  PROC DrawPart46()
    MoveL Offs(pOrigin,252.98,111.04,0.00),v40,z0,tPen\WObj:=wPaper;
    MoveL Offs(pOrigin,252.55,110.82,0.00),v40,fine,tPen\WObj:=wPaper;
    MoveL Offs(pOrigin,252.55,110.82,6.00),v60,z5,tPen\WObj:=wPaper;
    MoveL Offs(pOrigin,253.40,114.65,6.00),vTravel,z5,tPen\WObj:=wPaper;
    MoveL Offs(pOrigin,253.40,114.65,0.00),v60,z0,tPen\WObj:=wPaper;
    MoveL Offs(pOrigin,252.98,115.29,0.00),v40,z0,tPen\WObj:=wPaper;
    MoveL Offs(pOrigin,253.40,114.65,0.00),v40,fine,tPen\WObj:=wPaper;
    MoveL Offs(pOrigin,253.40,114.65,6.00),v60,z5,tPen\WObj:=wPaper;
    MoveL Offs(pOrigin,248.51,114.22,6.00),vTravel,z5,tPen\WObj:=wPaper;
    MoveL Offs(pOrigin,248.51,114.22,0.00),v60,z0,tPen\WObj:=wPaper;
    MoveL Offs(pOrigin,248.73,114.65,0.00),v40,z0,tPen\WObj:=wPaper;
    MoveL Offs(pOrigin,248.51,114.22,0.00),v40,fine,tPen\WObj:=wPaper;
    MoveL Offs(pOrigin,248.51,114.22,6.00),v60,z5,tPen\WObj:=wPaper;
    MoveL Offs(pOrigin,237.25,127.61,6.00),vTravel,z5,tPen\WObj:=wPaper;
    MoveL Offs(pOrigin,237.25,127.61,0.00),v60,z0,tPen\WObj:=wPaper;
    MoveL Offs(pOrigin,235.55,135.69,0.00),v40,fine,tPen\WObj:=wPaper;
    MoveL Offs(pOrigin,235.55,135.69,6.00),v60,z5,tPen\WObj:=wPaper;
    MoveL Offs(pOrigin,208.14,123.79,6.00),vTravel,z5,tPen\WObj:=wPaper;
    MoveL Offs(pOrigin,208.14,123.79,0.00),v60,z0,tPen\WObj:=wPaper;
    MoveL Offs(pOrigin,208.92,123.36,0.00),v40,z0,tPen\WObj:=wPaper;
    MoveL Offs(pOrigin,211.75,113.38,0.00),v40,z0,tPen\WObj:=wPaper;
    MoveL Offs(pOrigin,214.73,101.05,0.00),v40,z0,tPen\WObj:=wPaper;
    MoveL Offs(pOrigin,216.43,90.85,0.00),v40,z0,tPen\WObj:=wPaper;
    MoveL Offs(pOrigin,217.27,82.14,0.00),v40,z0,tPen\WObj:=wPaper;
    MoveL Offs(pOrigin,217.49,71.94,0.00),v40,z0,tPen\WObj:=wPaper;
    MoveL Offs(pOrigin,216.85,63.44,0.00),v40,z0,tPen\WObj:=wPaper;
    MoveL Offs(pOrigin,216.00,62.80,0.00),v40,z0,tPen\WObj:=wPaper;
    MoveL Offs(pOrigin,216.00,62.80,0.00),v40,z0,tPen\WObj:=wPaper;
    MoveL Offs(pOrigin,215.15,64.07,0.00),v40,z0,tPen\WObj:=wPaper;
    MoveL Offs(pOrigin,215.15,68.11,0.00),v40,z0,tPen\WObj:=wPaper;
    MoveL Offs(pOrigin,214.58,70.45,0.00),v40,z0,tPen\WObj:=wPaper;
    MoveL Offs(pOrigin,213.66,71.94,0.00),v40,z0,tPen\WObj:=wPaper;
    MoveL Offs(pOrigin,212.39,72.86,0.00),v40,z0,tPen\WObj:=wPaper;
    MoveL Offs(pOrigin,207.71,74.70,0.00),v40,z0,tPen\WObj:=wPaper;
    MoveL Offs(pOrigin,204.31,75.34,0.00),v40,z0,tPen\WObj:=wPaper;
    MoveL Offs(pOrigin,198.36,75.76,0.00),v40,z0,tPen\WObj:=wPaper;
    MoveL Offs(pOrigin,195.60,75.55,0.00),v40,z0,tPen\WObj:=wPaper;
    MoveL Offs(pOrigin,195.60,75.55,0.00),v40,z0,tPen\WObj:=wPaper;
    MoveL Offs(pOrigin,196.59,73.21,0.00),v40,z0,tPen\WObj:=wPaper;
    MoveL Offs(pOrigin,196.24,72.79,0.00),v40,z0,tPen\WObj:=wPaper;
    MoveL Offs(pOrigin,194.96,72.93,0.00),v40,z0,tPen\WObj:=wPaper;
    MoveL Offs(pOrigin,192.20,74.70,0.00),v40,z0,tPen\WObj:=wPaper;
    MoveL Offs(pOrigin,192.20,74.70,0.00),v40,z0,tPen\WObj:=wPaper;
    MoveL Offs(pOrigin,192.06,75.76,0.00),v40,z0,tPen\WObj:=wPaper;
    MoveL Offs(pOrigin,189.23,78.31,0.00),v40,z0,tPen\WObj:=wPaper;
    MoveL Offs(pOrigin,189.23,78.31,0.00),v40,z0,tPen\WObj:=wPaper;
    MoveL Offs(pOrigin,187.52,76.47,0.00),v40,z0,tPen\WObj:=wPaper;
    MoveL Offs(pOrigin,186.25,76.82,0.00),v40,fine,tPen\WObj:=wPaper;
    MoveL Offs(pOrigin,186.25,76.82,6.00),v60,z5,tPen\WObj:=wPaper;
    MoveL Offs(pOrigin,187.74,76.40,6.00),vTravel,z5,tPen\WObj:=wPaper;
    MoveL Offs(pOrigin,187.74,76.40,0.00),v60,z0,tPen\WObj:=wPaper;
    MoveL Offs(pOrigin,187.95,76.05,0.00),v40,z0,tPen\WObj:=wPaper;
    MoveL Offs(pOrigin,190.71,74.84,0.00),v40,z0,tPen\WObj:=wPaper;
    MoveL Offs(pOrigin,192.20,74.70,0.00),v40,fine,tPen\WObj:=wPaper;
    MoveL Offs(pOrigin,192.20,74.70,6.00),v60,z5,tPen\WObj:=wPaper;
    MoveL Offs(pOrigin,190.50,75.12,6.00),vTravel,z5,tPen\WObj:=wPaper;
    MoveL Offs(pOrigin,190.50,75.12,0.00),v60,z0,tPen\WObj:=wPaper;
    MoveL Offs(pOrigin,190.93,74.91,0.00),v40,z0,tPen\WObj:=wPaper;
    MoveL Offs(pOrigin,190.50,75.12,0.00),v40,z0,tPen\WObj:=wPaper;
    MoveL Offs(pOrigin,189.44,75.55,0.00),v40,z0,tPen\WObj:=wPaper;
    MoveL Offs(pOrigin,189.86,75.34,0.00),v40,z0,tPen\WObj:=wPaper;
    MoveL Offs(pOrigin,189.44,75.55,0.00),v40,fine,tPen\WObj:=wPaper;
    MoveL Offs(pOrigin,189.44,75.55,6.00),v60,z5,tPen\WObj:=wPaper;
    MoveL Offs(pOrigin,190.29,77.46,6.00),vTravel,z5,tPen\WObj:=wPaper;
    MoveL Offs(pOrigin,190.29,77.46,0.00),v60,z0,tPen\WObj:=wPaper;
    MoveL Offs(pOrigin,190.50,77.04,0.00),v40,z0,tPen\WObj:=wPaper;
    MoveL Offs(pOrigin,190.29,77.46,0.00),v40,z0,tPen\WObj:=wPaper;
    MoveL Offs(pOrigin,189.86,77.68,0.00),v40,z0,tPen\WObj:=wPaper;
    MoveL Offs(pOrigin,189.65,78.10,0.00),v40,z0,tPen\WObj:=wPaper;
    MoveL Offs(pOrigin,189.86,77.68,0.00),v40,fine,tPen\WObj:=wPaper;
    MoveL Offs(pOrigin,189.86,77.68,6.00),v60,z5,tPen\WObj:=wPaper;
    MoveL Offs(pOrigin,189.23,78.74,6.00),vTravel,z5,tPen\WObj:=wPaper;
    MoveL Offs(pOrigin,189.23,78.74,0.00),v60,z0,tPen\WObj:=wPaper;
    MoveL Offs(pOrigin,187.52,80.44,0.00),v40,z0,tPen\WObj:=wPaper;
    MoveL Offs(pOrigin,187.52,80.44,0.00),v40,z0,tPen\WObj:=wPaper;
    MoveL Offs(pOrigin,188.38,81.71,0.00),v40,z0,tPen\WObj:=wPaper;
    MoveL Offs(pOrigin,188.16,82.35,0.00),v40,z0,tPen\WObj:=wPaper;
    MoveL Offs(pOrigin,187.95,82.78,0.00),v40,z0,tPen\WObj:=wPaper;
    MoveL Offs(pOrigin,188.16,82.35,0.00),v40,z0,tPen\WObj:=wPaper;
    MoveL Offs(pOrigin,187.52,82.99,0.00),v40,z0,tPen\WObj:=wPaper;
    MoveL Offs(pOrigin,187.31,83.41,0.00),v40,z0,tPen\WObj:=wPaper;
    MoveL Offs(pOrigin,187.52,82.99,0.00),v40,fine,tPen\WObj:=wPaper;
    MoveL Offs(pOrigin,187.52,82.99,6.00),v60,z5,tPen\WObj:=wPaper;
    MoveL Offs(pOrigin,186.46,84.05,6.00),vTravel,z5,tPen\WObj:=wPaper;
    MoveL Offs(pOrigin,186.46,84.05,0.00),v60,z0,tPen\WObj:=wPaper;
    MoveL Offs(pOrigin,186.89,83.62,0.00),v40,z0,tPen\WObj:=wPaper;
    MoveL Offs(pOrigin,186.46,84.05,0.00),v40,z0,tPen\WObj:=wPaper;
    MoveL Offs(pOrigin,186.04,84.26,0.00),v40,z0,tPen\WObj:=wPaper;
    MoveL Offs(pOrigin,185.82,84.69,0.00),v40,z0,tPen\WObj:=wPaper;
    MoveL Offs(pOrigin,186.04,84.26,0.00),v40,fine,tPen\WObj:=wPaper;
    MoveL Offs(pOrigin,186.04,84.26,6.00),v60,z5,tPen\WObj:=wPaper;
    MoveL Offs(pOrigin,184.55,83.20,6.00),vTravel,z5,tPen\WObj:=wPaper;
    MoveL Offs(pOrigin,184.55,83.20,0.00),v60,z0,tPen\WObj:=wPaper;
    MoveL Offs(pOrigin,187.52,80.44,0.00),v40,fine,tPen\WObj:=wPaper;
    MoveL Offs(pOrigin,187.52,80.44,6.00),v60,z5,tPen\WObj:=wPaper;
    MoveL Offs(pOrigin,188.16,79.38,6.00),vTravel,z5,tPen\WObj:=wPaper;
    MoveL Offs(pOrigin,188.16,79.38,0.00),v60,z0,tPen\WObj:=wPaper;
    MoveL Offs(pOrigin,187.74,80.01,0.00),v40,z0,tPen\WObj:=wPaper;
    MoveL Offs(pOrigin,188.16,79.38,0.00),v40,fine,tPen\WObj:=wPaper;
    MoveL Offs(pOrigin,188.16,79.38,6.00),v60,z5,tPen\WObj:=wPaper;
    MoveL Offs(pOrigin,189.23,78.74,6.00),vTravel,z5,tPen\WObj:=wPaper;
    MoveL Offs(pOrigin,189.23,78.74,0.00),v60,z0,tPen\WObj:=wPaper;
    MoveL Offs(pOrigin,189.86,79.38,0.00),v40,z0,tPen\WObj:=wPaper;
    MoveL Offs(pOrigin,189.65,80.44,0.00),v40,z0,tPen\WObj:=wPaper;
    MoveL Offs(pOrigin,189.44,80.86,0.00),v40,z0,tPen\WObj:=wPaper;
    MoveL Offs(pOrigin,189.65,80.44,0.00),v40,fine,tPen\WObj:=wPaper;
    MoveL Offs(pOrigin,189.65,80.44,6.00),v60,z5,tPen\WObj:=wPaper;
    MoveL Offs(pOrigin,192.20,77.68,6.00),vTravel,z5,tPen\WObj:=wPaper;
    MoveL Offs(pOrigin,192.20,77.68,0.00),v60,z0,tPen\WObj:=wPaper;
    MoveL Offs(pOrigin,191.56,78.31,0.00),v40,z0,tPen\WObj:=wPaper;
    MoveL Offs(pOrigin,192.20,77.68,0.00),v40,fine,tPen\WObj:=wPaper;
    MoveL Offs(pOrigin,192.20,77.68,6.00),v60,z5,tPen\WObj:=wPaper;
    MoveL Offs(pOrigin,193.90,76.19,6.00),vTravel,z5,tPen\WObj:=wPaper;
    MoveL Offs(pOrigin,193.90,76.19,0.00),v60,z0,tPen\WObj:=wPaper;
    MoveL Offs(pOrigin,193.05,77.04,0.00),v40,z0,tPen\WObj:=wPaper;
    MoveL Offs(pOrigin,193.90,76.19,0.00),v40,fine,tPen\WObj:=wPaper;
    MoveL Offs(pOrigin,193.90,76.19,6.00),v60,z5,tPen\WObj:=wPaper;
    MoveL Offs(pOrigin,185.19,82.56,6.00),vTravel,z5,tPen\WObj:=wPaper;
    MoveL Offs(pOrigin,185.19,82.56,0.00),v60,z0,tPen\WObj:=wPaper;
    MoveL Offs(pOrigin,185.40,82.14,0.00),v40,z0,tPen\WObj:=wPaper;
  ENDPROC

  PROC DrawPart47()
    MoveL Offs(pOrigin,185.19,82.56,0.00),v40,fine,tPen\WObj:=wPaper;
    MoveL Offs(pOrigin,185.19,82.56,6.00),v60,z5,tPen\WObj:=wPaper;
    MoveL Offs(pOrigin,184.12,83.41,6.00),vTravel,z5,tPen\WObj:=wPaper;
    MoveL Offs(pOrigin,184.12,83.41,0.00),v60,z0,tPen\WObj:=wPaper;
    MoveL Offs(pOrigin,179.24,87.88,0.00),v40,z0,tPen\WObj:=wPaper;
    MoveL Offs(pOrigin,169.46,95.95,0.00),v40,z0,tPen\WObj:=wPaper;
    MoveL Offs(pOrigin,169.46,95.95,0.00),v40,z0,tPen\WObj:=wPaper;
    MoveL Offs(pOrigin,168.82,95.31,0.00),v40,fine,tPen\WObj:=wPaper;
    MoveL Offs(pOrigin,168.82,95.31,6.00),v60,z5,tPen\WObj:=wPaper;
    MoveL Offs(pOrigin,169.68,96.59,6.00),vTravel,z5,tPen\WObj:=wPaper;
    MoveL Offs(pOrigin,169.68,96.59,0.00),v60,z0,tPen\WObj:=wPaper;
    MoveL Offs(pOrigin,167.98,97.22,0.00),v40,z0,tPen\WObj:=wPaper;
    MoveL Offs(pOrigin,166.91,96.80,0.00),v40,z0,tPen\WObj:=wPaper;
    MoveL Offs(pOrigin,165.64,95.53,0.00),v40,fine,tPen\WObj:=wPaper;
    MoveL Offs(pOrigin,165.64,95.53,6.00),v60,z5,tPen\WObj:=wPaper;
    MoveL Offs(pOrigin,163.51,97.01,6.00),vTravel,z5,tPen\WObj:=wPaper;
    MoveL Offs(pOrigin,163.51,97.01,0.00),v60,z0,tPen\WObj:=wPaper;
    MoveL Offs(pOrigin,162.80,95.74,0.00),v40,z0,tPen\WObj:=wPaper;
    MoveL Offs(pOrigin,162.38,93.82,0.00),v40,z0,tPen\WObj:=wPaper;
    MoveL Offs(pOrigin,161.46,93.19,0.00),v40,z0,tPen\WObj:=wPaper;
    MoveL Offs(pOrigin,160.96,92.34,0.00),v40,z0,tPen\WObj:=wPaper;
    MoveL Offs(pOrigin,160.96,92.34,0.00),v40,z0,tPen\WObj:=wPaper;
    MoveL Offs(pOrigin,158.20,91.28,0.00),v40,z0,tPen\WObj:=wPaper;
    MoveL Offs(pOrigin,155.01,92.48,0.00),v40,z0,tPen\WObj:=wPaper;
    MoveL Offs(pOrigin,151.40,94.68,0.00),v40,fine,tPen\WObj:=wPaper;
    MoveL Offs(pOrigin,151.40,94.68,6.00),v60,z5,tPen\WObj:=wPaper;
    MoveL Offs(pOrigin,146.51,99.56,6.00),vTravel,z5,tPen\WObj:=wPaper;
    MoveL Offs(pOrigin,146.51,99.56,0.00),v60,z0,tPen\WObj:=wPaper;
    MoveL Offs(pOrigin,151.61,98.93,0.00),v40,z0,tPen\WObj:=wPaper;
    MoveL Offs(pOrigin,157.99,98.93,0.00),v40,z0,tPen\WObj:=wPaper;
    MoveL Offs(pOrigin,160.54,99.49,0.00),v40,z0,tPen\WObj:=wPaper;
    MoveL Offs(pOrigin,162.88,101.90,0.00),v40,z0,tPen\WObj:=wPaper;
    MoveL Offs(pOrigin,162.88,101.90,0.00),v40,z0,tPen\WObj:=wPaper;
    MoveL Offs(pOrigin,161.81,101.05,0.00),v40,fine,tPen\WObj:=wPaper;
    MoveL Offs(pOrigin,161.81,101.05,6.00),v60,z5,tPen\WObj:=wPaper;
    MoveL Offs(pOrigin,162.88,103.18,6.00),vTravel,z5,tPen\WObj:=wPaper;
    MoveL Offs(pOrigin,162.88,103.18,0.00),v60,z0,tPen\WObj:=wPaper;
    MoveL Offs(pOrigin,160.96,103.74,0.00),v40,z0,tPen\WObj:=wPaper;
    MoveL Offs(pOrigin,159.26,104.95,0.00),v40,z0,tPen\WObj:=wPaper;
    MoveL Offs(pOrigin,156.50,106.22,0.00),v40,z0,tPen\WObj:=wPaper;
    MoveL Offs(pOrigin,150.76,107.85,0.00),v40,fine,tPen\WObj:=wPaper;
    MoveL Offs(pOrigin,150.76,107.85,6.00),v60,z5,tPen\WObj:=wPaper;
    MoveL Offs(pOrigin,143.96,115.07,6.00),vTravel,z5,tPen\WObj:=wPaper;
    MoveL Offs(pOrigin,143.96,115.07,0.00),v60,z0,tPen\WObj:=wPaper;
    MoveL Offs(pOrigin,148.85,116.35,0.00),v40,z0,tPen\WObj:=wPaper;
    MoveL Offs(pOrigin,152.04,116.78,0.00),v40,z0,tPen\WObj:=wPaper;
    MoveL Offs(pOrigin,155.65,116.56,0.00),v40,z0,tPen\WObj:=wPaper;
    MoveL Offs(pOrigin,158.20,115.78,0.00),v40,z0,tPen\WObj:=wPaper;
    MoveL Offs(pOrigin,158.84,115.29,0.00),v40,z0,tPen\WObj:=wPaper;
    MoveL Offs(pOrigin,159.48,115.07,0.00),v40,z0,tPen\WObj:=wPaper;
    MoveL Offs(pOrigin,159.26,115.29,0.00),v40,z0,tPen\WObj:=wPaper;
    MoveL Offs(pOrigin,159.48,114.86,0.00),v40,z0,tPen\WObj:=wPaper;
    MoveL Offs(pOrigin,161.18,114.44,0.00),v40,fine,tPen\WObj:=wPaper;
    MoveL Offs(pOrigin,161.18,114.44,6.00),v60,z5,tPen\WObj:=wPaper;
    MoveL Offs(pOrigin,165.21,112.74,6.00),vTravel,z5,tPen\WObj:=wPaper;
    MoveL Offs(pOrigin,165.21,112.74,0.00),v60,z0,tPen\WObj:=wPaper;
    MoveL Offs(pOrigin,165.43,113.16,0.00),v40,z0,tPen\WObj:=wPaper;
    MoveL Offs(pOrigin,165.21,112.74,0.00),v40,z0,tPen\WObj:=wPaper;
    MoveL Offs(pOrigin,165.64,113.59,0.00),v40,z0,tPen\WObj:=wPaper;
    MoveL Offs(pOrigin,165.85,114.01,0.00),v40,z0,tPen\WObj:=wPaper;
    MoveL Offs(pOrigin,165.64,113.59,0.00),v40,fine,tPen\WObj:=wPaper;
    MoveL Offs(pOrigin,165.64,113.59,6.00),v60,z5,tPen\WObj:=wPaper;
    MoveL Offs(pOrigin,166.27,114.65,6.00),vTravel,z5,tPen\WObj:=wPaper;
    MoveL Offs(pOrigin,166.27,114.65,0.00),v60,z0,tPen\WObj:=wPaper;
    MoveL Offs(pOrigin,166.49,115.07,0.00),v40,z0,tPen\WObj:=wPaper;
    MoveL Offs(pOrigin,166.27,114.65,0.00),v40,fine,tPen\WObj:=wPaper;
    MoveL Offs(pOrigin,166.27,114.65,6.00),v60,z5,tPen\WObj:=wPaper;
    MoveL Offs(pOrigin,169.25,113.38,6.00),vTravel,z5,tPen\WObj:=wPaper;
    MoveL Offs(pOrigin,169.25,113.38,0.00),v60,z0,tPen\WObj:=wPaper;
    MoveL Offs(pOrigin,169.68,114.01,0.00),v40,z0,tPen\WObj:=wPaper;
    MoveL Offs(pOrigin,169.25,113.38,0.00),v40,fine,tPen\WObj:=wPaper;
    MoveL Offs(pOrigin,169.25,113.38,6.00),v60,z5,tPen\WObj:=wPaper;
    MoveL Offs(pOrigin,168.19,111.89,6.00),vTravel,z5,tPen\WObj:=wPaper;
    MoveL Offs(pOrigin,168.19,111.89,0.00),v60,z0,tPen\WObj:=wPaper;
    MoveL Offs(pOrigin,168.61,112.53,0.00),v40,z0,tPen\WObj:=wPaper;
    MoveL Offs(pOrigin,168.19,111.89,0.00),v40,fine,tPen\WObj:=wPaper;
    MoveL Offs(pOrigin,168.19,111.89,6.00),v60,z5,tPen\WObj:=wPaper;
    MoveL Offs(pOrigin,166.70,109.76,6.00),vTravel,z5,tPen\WObj:=wPaper;
    MoveL Offs(pOrigin,166.70,109.76,0.00),v60,z0,tPen\WObj:=wPaper;
    MoveL Offs(pOrigin,167.12,110.40,0.00),v40,z0,tPen\WObj:=wPaper;
    MoveL Offs(pOrigin,166.70,109.76,0.00),v40,fine,tPen\WObj:=wPaper;
    MoveL Offs(pOrigin,166.70,109.76,6.00),v60,z5,tPen\WObj:=wPaper;
    MoveL Offs(pOrigin,163.09,104.24,6.00),vTravel,z5,tPen\WObj:=wPaper;
    MoveL Offs(pOrigin,163.09,104.24,0.00),v60,z0,tPen\WObj:=wPaper;
    MoveL Offs(pOrigin,162.66,105.72,0.00),v40,z0,tPen\WObj:=wPaper;
    MoveL Offs(pOrigin,162.73,108.06,0.00),v40,z0,tPen\WObj:=wPaper;
    MoveL Offs(pOrigin,163.58,108.91,0.00),v40,z0,tPen\WObj:=wPaper;
    MoveL Offs(pOrigin,164.72,111.68,0.00),v40,z0,tPen\WObj:=wPaper;
    MoveL Offs(pOrigin,167.90,117.20,0.00),v40,z0,tPen\WObj:=wPaper;
    MoveL Offs(pOrigin,171.80,122.72,0.00),v40,z0,tPen\WObj:=wPaper;
    MoveL Offs(pOrigin,171.38,122.30,0.00),v40,z0,tPen\WObj:=wPaper;
    MoveL Offs(pOrigin,171.80,122.72,0.00),v40,z0,tPen\WObj:=wPaper;
    MoveL Offs(pOrigin,171.38,122.30,0.00),v40,fine,tPen\WObj:=wPaper;
    MoveL Offs(pOrigin,171.38,122.30,6.00),v60,z5,tPen\WObj:=wPaper;
    MoveL Offs(pOrigin,168.40,118.05,6.00),vTravel,z5,tPen\WObj:=wPaper;
    MoveL Offs(pOrigin,168.40,118.05,0.00),v60,z0,tPen\WObj:=wPaper;
    MoveL Offs(pOrigin,168.82,118.69,0.00),v40,z0,tPen\WObj:=wPaper;
    MoveL Offs(pOrigin,168.40,118.05,0.00),v40,fine,tPen\WObj:=wPaper;
    MoveL Offs(pOrigin,168.40,118.05,6.00),v60,z5,tPen\WObj:=wPaper;
    MoveL Offs(pOrigin,159.90,124.00,6.00),vTravel,z5,tPen\WObj:=wPaper;
    MoveL Offs(pOrigin,159.90,124.00,0.00),v60,z0,tPen\WObj:=wPaper;
    MoveL Offs(pOrigin,158.62,124.28,0.00),v40,z0,tPen\WObj:=wPaper;
    MoveL Offs(pOrigin,153.74,128.11,0.00),v40,z0,tPen\WObj:=wPaper;
    MoveL Offs(pOrigin,148.64,130.87,0.00),v40,z0,tPen\WObj:=wPaper;
    MoveL Offs(pOrigin,143.75,132.78,0.00),v40,z0,tPen\WObj:=wPaper;
    MoveL Offs(pOrigin,140.56,133.56,0.00),v40,fine,tPen\WObj:=wPaper;
    MoveL Offs(pOrigin,140.56,133.56,6.00),v60,z5,tPen\WObj:=wPaper;
    MoveL Offs(pOrigin,135.46,137.81,6.00),vTravel,z5,tPen\WObj:=wPaper;
    MoveL Offs(pOrigin,135.46,137.81,0.00),v60,z0,tPen\WObj:=wPaper;
    MoveL Offs(pOrigin,137.59,137.81,0.00),v40,z0,tPen\WObj:=wPaper;
    MoveL Offs(pOrigin,141.20,137.18,0.00),v40,z0,tPen\WObj:=wPaper;
    MoveL Offs(pOrigin,147.36,135.33,0.00),v40,z0,tPen\WObj:=wPaper;
    MoveL Offs(pOrigin,151.82,133.21,0.00),v40,z0,tPen\WObj:=wPaper;
    MoveL Offs(pOrigin,155.44,130.80,0.00),v40,z0,tPen\WObj:=wPaper;
    MoveL Offs(pOrigin,155.86,130.59,0.00),v40,z0,tPen\WObj:=wPaper;
    MoveL Offs(pOrigin,157.77,128.82,0.00),v40,z0,tPen\WObj:=wPaper;
    MoveL Offs(pOrigin,159.05,128.46,0.00),v40,fine,tPen\WObj:=wPaper;
    MoveL Offs(pOrigin,159.05,128.46,6.00),v60,z5,tPen\WObj:=wPaper;
    MoveL Offs(pOrigin,157.14,129.31,6.00),vTravel,z5,tPen\WObj:=wPaper;
    MoveL Offs(pOrigin,157.14,129.31,0.00),v60,z0,tPen\WObj:=wPaper;
  ENDPROC

  PROC DrawPart48()
    MoveL Offs(pOrigin,156.93,129.74,0.00),v40,z0,tPen\WObj:=wPaper;
    MoveL Offs(pOrigin,157.14,129.31,0.00),v40,fine,tPen\WObj:=wPaper;
    MoveL Offs(pOrigin,157.14,129.31,6.00),v60,z5,tPen\WObj:=wPaper;
    MoveL Offs(pOrigin,156.29,126.34,6.00),vTravel,z5,tPen\WObj:=wPaper;
    MoveL Offs(pOrigin,156.29,126.34,0.00),v60,z0,tPen\WObj:=wPaper;
    MoveL Offs(pOrigin,156.71,126.12,0.00),v40,z0,tPen\WObj:=wPaper;
    MoveL Offs(pOrigin,156.29,126.34,0.00),v40,fine,tPen\WObj:=wPaper;
    MoveL Offs(pOrigin,156.29,126.34,6.00),v60,z5,tPen\WObj:=wPaper;
    MoveL Offs(pOrigin,157.56,125.06,6.00),vTravel,z5,tPen\WObj:=wPaper;
    MoveL Offs(pOrigin,157.56,125.06,0.00),v60,z0,tPen\WObj:=wPaper;
    MoveL Offs(pOrigin,157.35,125.49,0.00),v40,z0,tPen\WObj:=wPaper;
    MoveL Offs(pOrigin,157.56,125.06,0.00),v40,fine,tPen\WObj:=wPaper;
    MoveL Offs(pOrigin,157.56,125.06,6.00),v60,z5,tPen\WObj:=wPaper;
    MoveL Offs(pOrigin,157.35,119.75,6.00),vTravel,z5,tPen\WObj:=wPaper;
    MoveL Offs(pOrigin,157.35,119.75,0.00),v60,z0,tPen\WObj:=wPaper;
    MoveL Offs(pOrigin,152.46,119.96,0.00),v40,z0,tPen\WObj:=wPaper;
    MoveL Offs(pOrigin,149.06,119.54,0.00),v40,z0,tPen\WObj:=wPaper;
    MoveL Offs(pOrigin,143.32,118.26,0.00),v40,z0,tPen\WObj:=wPaper;
    MoveL Offs(pOrigin,138.65,116.56,0.00),v40,fine,tPen\WObj:=wPaper;
    MoveL Offs(pOrigin,138.65,116.56,6.00),v60,z5,tPen\WObj:=wPaper;
    MoveL Offs(pOrigin,131.64,124.00,6.00),vTravel,z5,tPen\WObj:=wPaper;
    MoveL Offs(pOrigin,131.64,124.00,0.00),v60,z0,tPen\WObj:=wPaper;
    MoveL Offs(pOrigin,130.36,122.51,0.00),v40,z0,tPen\WObj:=wPaper;
    MoveL Offs(pOrigin,127.60,120.53,0.00),v40,z0,tPen\WObj:=wPaper;
    MoveL Offs(pOrigin,117.40,114.65,0.00),v40,fine,tPen\WObj:=wPaper;
    MoveL Offs(pOrigin,117.40,114.65,6.00),v60,z5,tPen\WObj:=wPaper;
    MoveL Offs(pOrigin,118.89,130.16,6.00),vTravel,z5,tPen\WObj:=wPaper;
    MoveL Offs(pOrigin,118.89,130.16,0.00),v60,z0,tPen\WObj:=wPaper;
    MoveL Offs(pOrigin,119.10,130.59,0.00),v40,z0,tPen\WObj:=wPaper;
    MoveL Offs(pOrigin,118.89,130.16,0.00),v40,fine,tPen\WObj:=wPaper;
    MoveL Offs(pOrigin,118.89,130.16,6.00),v60,z5,tPen\WObj:=wPaper;
    MoveL Offs(pOrigin,123.78,133.14,6.00),vTravel,z5,tPen\WObj:=wPaper;
    MoveL Offs(pOrigin,123.78,133.14,0.00),v60,z0,tPen\WObj:=wPaper;
    MoveL Offs(pOrigin,136.74,131.01,0.00),v40,z0,tPen\WObj:=wPaper;
    MoveL Offs(pOrigin,146.73,128.04,0.00),v40,z0,tPen\WObj:=wPaper;
    MoveL Offs(pOrigin,149.49,126.76,0.00),v40,fine,tPen\WObj:=wPaper;
    MoveL Offs(pOrigin,149.49,126.76,6.00),v60,z5,tPen\WObj:=wPaper;
    MoveL Offs(pOrigin,150.55,129.95,6.00),vTravel,z5,tPen\WObj:=wPaper;
    MoveL Offs(pOrigin,150.55,129.95,0.00),v60,z0,tPen\WObj:=wPaper;
    MoveL Offs(pOrigin,150.98,129.74,0.00),v40,z0,tPen\WObj:=wPaper;
    MoveL Offs(pOrigin,150.55,129.95,0.00),v40,z0,tPen\WObj:=wPaper;
    MoveL Offs(pOrigin,149.70,130.38,0.00),v40,z0,tPen\WObj:=wPaper;
    MoveL Offs(pOrigin,150.12,130.16,0.00),v40,z0,tPen\WObj:=wPaper;
    MoveL Offs(pOrigin,149.70,130.38,0.00),v40,fine,tPen\WObj:=wPaper;
    MoveL Offs(pOrigin,149.70,130.38,6.00),v60,z5,tPen\WObj:=wPaper;
    MoveL Offs(pOrigin,155.65,135.69,6.00),vTravel,z5,tPen\WObj:=wPaper;
    MoveL Offs(pOrigin,155.65,135.69,0.00),v60,z0,tPen\WObj:=wPaper;
    MoveL Offs(pOrigin,157.14,135.69,0.00),v40,z0,tPen\WObj:=wPaper;
    MoveL Offs(pOrigin,157.35,137.18,0.00),v40,z0,tPen\WObj:=wPaper;
    MoveL Offs(pOrigin,152.68,152.26,0.00),v40,z0,tPen\WObj:=wPaper;
    MoveL Offs(pOrigin,150.12,159.27,0.00),v40,fine,tPen\WObj:=wPaper;
    MoveL Offs(pOrigin,150.12,159.27,6.00),v60,z5,tPen\WObj:=wPaper;
    MoveL Offs(pOrigin,145.66,165.44,6.00),vTravel,z5,tPen\WObj:=wPaper;
    MoveL Offs(pOrigin,145.66,165.44,0.00),v60,z0,tPen\WObj:=wPaper;
    MoveL Offs(pOrigin,145.45,165.86,0.00),v40,z0,tPen\WObj:=wPaper;
    MoveL Offs(pOrigin,145.66,165.44,0.00),v40,z0,tPen\WObj:=wPaper;
    MoveL Offs(pOrigin,145.24,166.29,0.00),v40,z0,tPen\WObj:=wPaper;
    MoveL Offs(pOrigin,145.02,166.71,0.00),v40,z0,tPen\WObj:=wPaper;
    MoveL Offs(pOrigin,145.24,166.29,0.00),v40,z0,tPen\WObj:=wPaper;
    MoveL Offs(pOrigin,144.81,167.14,0.00),v40,z0,tPen\WObj:=wPaper;
    MoveL Offs(pOrigin,144.60,167.56,0.00),v40,z0,tPen\WObj:=wPaper;
    MoveL Offs(pOrigin,144.81,167.14,0.00),v40,z0,tPen\WObj:=wPaper;
    MoveL Offs(pOrigin,144.39,167.99,0.00),v40,z0,tPen\WObj:=wPaper;
    MoveL Offs(pOrigin,144.18,168.41,0.00),v40,z0,tPen\WObj:=wPaper;
    MoveL Offs(pOrigin,144.39,167.99,0.00),v40,fine,tPen\WObj:=wPaper;
    MoveL Offs(pOrigin,144.39,167.99,6.00),v60,z5,tPen\WObj:=wPaper;
    MoveL Offs(pOrigin,144.81,148.86,6.00),vTravel,z5,tPen\WObj:=wPaper;
    MoveL Offs(pOrigin,144.81,148.86,0.00),v60,z0,tPen\WObj:=wPaper;
    MoveL Offs(pOrigin,145.02,148.44,0.00),v40,z0,tPen\WObj:=wPaper;
    MoveL Offs(pOrigin,144.81,148.86,0.00),v40,fine,tPen\WObj:=wPaper;
    MoveL Offs(pOrigin,144.81,148.86,6.00),v60,z5,tPen\WObj:=wPaper;
    MoveL Offs(pOrigin,145.66,147.80,6.00),vTravel,z5,tPen\WObj:=wPaper;
    MoveL Offs(pOrigin,145.66,147.80,0.00),v60,z0,tPen\WObj:=wPaper;
    MoveL Offs(pOrigin,145.45,148.23,0.00),v40,z0,tPen\WObj:=wPaper;
    MoveL Offs(pOrigin,145.66,147.80,0.00),v40,z0,tPen\WObj:=wPaper;
    MoveL Offs(pOrigin,146.30,147.16,0.00),v40,z0,tPen\WObj:=wPaper;
    MoveL Offs(pOrigin,146.09,147.59,0.00),v40,z0,tPen\WObj:=wPaper;
    MoveL Offs(pOrigin,146.30,147.16,0.00),v40,z0,tPen\WObj:=wPaper;
    MoveL Offs(pOrigin,146.73,146.95,0.00),v40,z0,tPen\WObj:=wPaper;
    MoveL Offs(pOrigin,146.94,146.52,0.00),v40,z0,tPen\WObj:=wPaper;
    MoveL Offs(pOrigin,146.73,146.95,0.00),v40,fine,tPen\WObj:=wPaper;
    MoveL Offs(pOrigin,146.73,146.95,6.00),v60,z5,tPen\WObj:=wPaper;
    MoveL Offs(pOrigin,147.57,145.89,6.00),vTravel,z5,tPen\WObj:=wPaper;
    MoveL Offs(pOrigin,147.57,145.89,0.00),v60,z0,tPen\WObj:=wPaper;
    MoveL Offs(pOrigin,147.36,146.31,0.00),v40,z0,tPen\WObj:=wPaper;
    MoveL Offs(pOrigin,147.57,145.89,0.00),v40,z0,tPen\WObj:=wPaper;
    MoveL Offs(pOrigin,148.21,145.25,0.00),v40,z0,tPen\WObj:=wPaper;
    MoveL Offs(pOrigin,148.00,145.68,0.00),v40,z0,tPen\WObj:=wPaper;
    MoveL Offs(pOrigin,148.21,145.25,0.00),v40,fine,tPen\WObj:=wPaper;
    MoveL Offs(pOrigin,148.21,145.25,6.00),v60,z5,tPen\WObj:=wPaper;
    MoveL Offs(pOrigin,149.91,143.34,6.00),vTravel,z5,tPen\WObj:=wPaper;
    MoveL Offs(pOrigin,149.91,143.34,0.00),v60,z0,tPen\WObj:=wPaper;
    MoveL Offs(pOrigin,149.70,143.76,0.00),v40,z0,tPen\WObj:=wPaper;
    MoveL Offs(pOrigin,149.91,143.34,0.00),v40,fine,tPen\WObj:=wPaper;
    MoveL Offs(pOrigin,149.91,143.34,6.00),v60,z5,tPen\WObj:=wPaper;
    MoveL Offs(pOrigin,151.40,141.85,6.00),vTravel,z5,tPen\WObj:=wPaper;
    MoveL Offs(pOrigin,151.40,141.85,0.00),v60,z0,tPen\WObj:=wPaper;
    MoveL Offs(pOrigin,151.61,141.43,0.00),v40,z0,tPen\WObj:=wPaper;
    MoveL Offs(pOrigin,151.40,141.85,0.00),v40,fine,tPen\WObj:=wPaper;
    MoveL Offs(pOrigin,151.40,141.85,6.00),v60,z5,tPen\WObj:=wPaper;
    MoveL Offs(pOrigin,152.68,140.15,6.00),vTravel,z5,tPen\WObj:=wPaper;
    MoveL Offs(pOrigin,152.68,140.15,0.00),v60,z0,tPen\WObj:=wPaper;
    MoveL Offs(pOrigin,152.46,140.57,0.00),v40,z0,tPen\WObj:=wPaper;
    MoveL Offs(pOrigin,152.68,140.15,0.00),v40,fine,tPen\WObj:=wPaper;
    MoveL Offs(pOrigin,152.68,140.15,6.00),v60,z5,tPen\WObj:=wPaper;
    MoveL Offs(pOrigin,153.52,139.30,6.00),vTravel,z5,tPen\WObj:=wPaper;
    MoveL Offs(pOrigin,153.52,139.30,0.00),v60,z0,tPen\WObj:=wPaper;
    MoveL Offs(pOrigin,153.74,138.88,0.00),v40,z0,tPen\WObj:=wPaper;
    MoveL Offs(pOrigin,153.52,139.30,0.00),v40,fine,tPen\WObj:=wPaper;
    MoveL Offs(pOrigin,153.52,139.30,6.00),v60,z5,tPen\WObj:=wPaper;
    MoveL Offs(pOrigin,154.80,137.60,6.00),vTravel,z5,tPen\WObj:=wPaper;
    MoveL Offs(pOrigin,154.80,137.60,0.00),v60,z0,tPen\WObj:=wPaper;
    MoveL Offs(pOrigin,154.59,138.02,0.00),v40,z0,tPen\WObj:=wPaper;
    MoveL Offs(pOrigin,154.80,137.60,0.00),v40,fine,tPen\WObj:=wPaper;
    MoveL Offs(pOrigin,154.80,137.60,6.00),v60,z5,tPen\WObj:=wPaper;
    MoveL Offs(pOrigin,155.65,135.69,6.00),vTravel,z5,tPen\WObj:=wPaper;
    MoveL Offs(pOrigin,155.65,135.69,0.00),v60,z0,tPen\WObj:=wPaper;
    MoveL Offs(pOrigin,154.16,136.11,0.00),v40,z0,tPen\WObj:=wPaper;
    MoveL Offs(pOrigin,147.15,141.43,0.00),v40,z0,tPen\WObj:=wPaper;
    MoveL Offs(pOrigin,146.51,141.64,0.00),v40,z0,tPen\WObj:=wPaper;
  ENDPROC

  PROC DrawPart49()
    MoveL Offs(pOrigin,145.66,142.35,0.00),v40,z0,tPen\WObj:=wPaper;
    MoveL Offs(pOrigin,140.77,144.61,0.00),v40,fine,tPen\WObj:=wPaper;
    MoveL Offs(pOrigin,140.77,144.61,6.00),v60,z5,tPen\WObj:=wPaper;
    MoveL Offs(pOrigin,126.32,138.88,6.00),vTravel,z5,tPen\WObj:=wPaper;
    MoveL Offs(pOrigin,126.32,138.88,0.00),v60,z0,tPen\WObj:=wPaper;
    MoveL Offs(pOrigin,126.54,139.30,0.00),v40,z0,tPen\WObj:=wPaper;
    MoveL Offs(pOrigin,126.32,138.88,0.00),v40,fine,tPen\WObj:=wPaper;
    MoveL Offs(pOrigin,126.32,138.88,6.00),v60,z5,tPen\WObj:=wPaper;
    MoveL Offs(pOrigin,133.12,96.16,6.00),vTravel,z5,tPen\WObj:=wPaper;
    MoveL Offs(pOrigin,133.12,96.16,0.00),v60,z0,tPen\WObj:=wPaper;
    MoveL Offs(pOrigin,138.44,95.31,0.00),v40,z0,tPen\WObj:=wPaper;
    MoveL Offs(pOrigin,142.26,93.90,0.00),v40,z0,tPen\WObj:=wPaper;
    MoveL Offs(pOrigin,145.88,91.98,0.00),v40,z0,tPen\WObj:=wPaper;
    MoveL Offs(pOrigin,150.55,88.51,0.00),v40,z0,tPen\WObj:=wPaper;
    MoveL Offs(pOrigin,152.46,86.60,0.00),v40,z0,tPen\WObj:=wPaper;
    MoveL Offs(pOrigin,157.14,80.22,0.00),v40,fine,tPen\WObj:=wPaper;
    MoveL Offs(pOrigin,157.14,80.22,6.00),v60,z5,tPen\WObj:=wPaper;
    MoveL Offs(pOrigin,158.84,77.25,6.00),vTravel,z5,tPen\WObj:=wPaper;
    MoveL Offs(pOrigin,158.84,77.25,0.00),v60,z0,tPen\WObj:=wPaper;
    MoveL Offs(pOrigin,159.48,76.75,0.00),v40,z0,tPen\WObj:=wPaper;
    MoveL Offs(pOrigin,169.04,73.43,0.00),v40,z0,tPen\WObj:=wPaper;
    MoveL Offs(pOrigin,169.04,73.43,0.00),v40,z0,tPen\WObj:=wPaper;
    MoveL Offs(pOrigin,168.68,75.55,0.00),v40,z0,tPen\WObj:=wPaper;
    MoveL Offs(pOrigin,166.84,79.38,0.00),v40,z0,tPen\WObj:=wPaper;
    MoveL Offs(pOrigin,165.00,84.47,0.00),v40,z0,tPen\WObj:=wPaper;
    MoveL Offs(pOrigin,163.09,92.76,0.00),v40,z0,tPen\WObj:=wPaper;
    MoveL Offs(pOrigin,162.45,93.61,0.00),v40,fine,tPen\WObj:=wPaper;
    MoveL Offs(pOrigin,162.45,93.61,6.00),v60,z5,tPen\WObj:=wPaper;
    MoveL Offs(pOrigin,160.96,92.34,6.00),vTravel,z5,tPen\WObj:=wPaper;
    MoveL Offs(pOrigin,160.96,92.34,0.00),v60,z0,tPen\WObj:=wPaper;
    MoveL Offs(pOrigin,161.18,89.36,0.00),v40,z0,tPen\WObj:=wPaper;
    MoveL Offs(pOrigin,160.75,84.05,0.00),v40,z0,tPen\WObj:=wPaper;
    MoveL Offs(pOrigin,158.98,77.68,0.00),v40,z0,tPen\WObj:=wPaper;
    MoveL Offs(pOrigin,158.41,77.25,0.00),v40,z0,tPen\WObj:=wPaper;
    MoveL Offs(pOrigin,150.12,79.73,0.00),v40,z0,tPen\WObj:=wPaper;
    MoveL Offs(pOrigin,143.75,82.63,0.00),v40,z0,tPen\WObj:=wPaper;
    MoveL Offs(pOrigin,142.90,83.98,0.00),v40,z0,tPen\WObj:=wPaper;
    MoveL Offs(pOrigin,139.93,85.61,0.00),v40,z0,tPen\WObj:=wPaper;
    MoveL Offs(pOrigin,139.29,86.53,0.00),v40,z0,tPen\WObj:=wPaper;
    MoveL Offs(pOrigin,138.01,87.31,0.00),v40,z0,tPen\WObj:=wPaper;
    MoveL Offs(pOrigin,135.25,88.44,0.00),v40,z0,tPen\WObj:=wPaper;
    MoveL Offs(pOrigin,132.49,90.07,0.00),v40,z0,tPen\WObj:=wPaper;
    MoveL Offs(pOrigin,130.79,90.43,0.00),v40,z0,tPen\WObj:=wPaper;
    MoveL Offs(pOrigin,130.79,90.43,0.00),v40,z0,tPen\WObj:=wPaper;
    MoveL Offs(pOrigin,130.15,89.57,0.00),v40,z0,tPen\WObj:=wPaper;
    MoveL Offs(pOrigin,124.84,89.79,0.00),v40,z0,tPen\WObj:=wPaper;
    MoveL Offs(pOrigin,120.80,88.80,0.00),v40,z0,tPen\WObj:=wPaper;
    MoveL Offs(pOrigin,116.12,86.67,0.00),v40,z0,tPen\WObj:=wPaper;
    MoveL Offs(pOrigin,111.88,83.62,0.00),v40,z0,tPen\WObj:=wPaper;
    MoveL Offs(pOrigin,108.69,80.44,0.00),v40,z0,tPen\WObj:=wPaper;
    MoveL Offs(pOrigin,104.58,74.91,0.00),v40,z0,tPen\WObj:=wPaper;
    MoveL Offs(pOrigin,101.18,68.54,0.00),v40,z0,tPen\WObj:=wPaper;
    MoveL Offs(pOrigin,99.97,65.56,0.00),v40,z0,tPen\WObj:=wPaper;
    MoveL Offs(pOrigin,99.97,64.71,0.00),v40,z0,tPen\WObj:=wPaper;
    MoveL Offs(pOrigin,99.97,64.71,0.00),v40,z0,tPen\WObj:=wPaper;
    MoveL Offs(pOrigin,100.61,64.93,0.00),v40,z0,tPen\WObj:=wPaper;
    MoveL Offs(pOrigin,103.80,67.69,0.00),v40,z0,tPen\WObj:=wPaper;
    MoveL Offs(pOrigin,106.78,70.66,0.00),v40,z0,tPen\WObj:=wPaper;
    MoveL Offs(pOrigin,111.88,77.04,0.00),v40,z0,tPen\WObj:=wPaper;
    MoveL Offs(pOrigin,115.49,79.87,0.00),v40,z0,tPen\WObj:=wPaper;
    MoveL Offs(pOrigin,118.25,81.36,0.00),v40,z0,tPen\WObj:=wPaper;
    MoveL Offs(pOrigin,122.50,82.78,0.00),v40,z0,tPen\WObj:=wPaper;
    MoveL Offs(pOrigin,125.69,83.41,0.00),v40,z0,tPen\WObj:=wPaper;
    MoveL Offs(pOrigin,128.24,83.41,0.00),v40,z0,tPen\WObj:=wPaper;
    MoveL Offs(pOrigin,128.24,83.41,0.00),v40,z0,tPen\WObj:=wPaper;
    MoveL Offs(pOrigin,134.19,83.62,0.00),v40,z0,tPen\WObj:=wPaper;
    MoveL Offs(pOrigin,141.84,82.35,0.00),v40,z0,tPen\WObj:=wPaper;
    MoveL Offs(pOrigin,143.54,82.56,0.00),v40,fine,tPen\WObj:=wPaper;
    MoveL Offs(pOrigin,143.54,82.56,6.00),v60,z5,tPen\WObj:=wPaper;
    MoveL Offs(pOrigin,139.71,85.54,6.00),vTravel,z5,tPen\WObj:=wPaper;
    MoveL Offs(pOrigin,139.71,85.54,0.00),v60,z0,tPen\WObj:=wPaper;
    MoveL Offs(pOrigin,138.65,85.32,0.00),v40,z0,tPen\WObj:=wPaper;
    MoveL Offs(pOrigin,135.53,87.03,0.00),v40,z0,tPen\WObj:=wPaper;
    MoveL Offs(pOrigin,135.25,88.30,0.00),v40,fine,tPen\WObj:=wPaper;
    MoveL Offs(pOrigin,135.25,88.30,6.00),v60,z5,tPen\WObj:=wPaper;
    MoveL Offs(pOrigin,130.79,90.43,6.00),vTravel,z5,tPen\WObj:=wPaper;
    MoveL Offs(pOrigin,130.79,90.43,0.00),v60,z0,tPen\WObj:=wPaper;
    MoveL Offs(pOrigin,130.57,90.85,0.00),v40,z0,tPen\WObj:=wPaper;
    MoveL Offs(pOrigin,127.81,91.91,0.00),v40,z0,tPen\WObj:=wPaper;
    MoveL Offs(pOrigin,121.01,93.40,0.00),v40,z0,tPen\WObj:=wPaper;
    MoveL Offs(pOrigin,115.70,93.40,0.00),v40,z0,tPen\WObj:=wPaper;
    MoveL Offs(pOrigin,112.51,92.97,0.00),v40,z0,tPen\WObj:=wPaper;
    MoveL Offs(pOrigin,106.14,90.85,0.00),v40,fine,tPen\WObj:=wPaper;
    MoveL Offs(pOrigin,106.14,90.85,6.00),v60,z5,tPen\WObj:=wPaper;
    MoveL Offs(pOrigin,104.01,94.68,6.00),vTravel,z5,tPen\WObj:=wPaper;
    MoveL Offs(pOrigin,104.01,94.68,0.00),v60,z0,tPen\WObj:=wPaper;
    MoveL Offs(pOrigin,102.53,92.97,0.00),v40,z0,tPen\WObj:=wPaper;
    MoveL Offs(pOrigin,100.40,91.28,0.00),v40,z0,tPen\WObj:=wPaper;
    MoveL Offs(pOrigin,98.42,88.51,0.00),v40,z0,tPen\WObj:=wPaper;
    MoveL Offs(pOrigin,95.80,82.14,0.00),v40,z0,tPen\WObj:=wPaper;
    MoveL Offs(pOrigin,91.40,74.70,0.00),v40,z0,tPen\WObj:=wPaper;
    MoveL Offs(pOrigin,90.20,71.09,0.00),v40,z0,tPen\WObj:=wPaper;
    MoveL Offs(pOrigin,89.99,69.60,0.00),v40,z0,tPen\WObj:=wPaper;
    MoveL Offs(pOrigin,90.20,63.44,0.00),v40,z0,tPen\WObj:=wPaper;
    MoveL Offs(pOrigin,92.18,56.21,0.00),v40,z0,tPen\WObj:=wPaper;
    MoveL Offs(pOrigin,92.96,55.58,0.00),v40,fine,tPen\WObj:=wPaper;
    MoveL Offs(pOrigin,92.96,55.58,6.00),v60,z5,tPen\WObj:=wPaper;
    MoveL Offs(pOrigin,93.81,52.39,6.00),vTravel,z5,tPen\WObj:=wPaper;
    MoveL Offs(pOrigin,93.81,52.39,0.00),v60,z0,tPen\WObj:=wPaper;
    MoveL Offs(pOrigin,94.24,52.60,0.00),v40,z0,tPen\WObj:=wPaper;
    MoveL Offs(pOrigin,93.81,52.39,0.00),v40,z0,tPen\WObj:=wPaper;
    MoveL Offs(pOrigin,93.18,51.96,0.00),v40,z0,tPen\WObj:=wPaper;
    MoveL Offs(pOrigin,93.18,55.58,0.00),v40,z0,tPen\WObj:=wPaper;
    MoveL Offs(pOrigin,93.88,56.42,0.00),v40,z0,tPen\WObj:=wPaper;
    MoveL Offs(pOrigin,95.23,60.25,0.00),v40,z0,tPen\WObj:=wPaper;
    MoveL Offs(pOrigin,98.49,66.84,0.00),v40,fine,tPen\WObj:=wPaper;
    MoveL Offs(pOrigin,98.49,66.84,6.00),v60,z5,tPen\WObj:=wPaper;
    MoveL Offs(pOrigin,99.97,64.71,6.00),vTravel,z5,tPen\WObj:=wPaper;
    MoveL Offs(pOrigin,99.97,64.71,0.00),v60,z0,tPen\WObj:=wPaper;
    MoveL Offs(pOrigin,97.35,59.83,0.00),v40,z0,tPen\WObj:=wPaper;
    MoveL Offs(pOrigin,94.52,52.81,0.00),v40,z0,tPen\WObj:=wPaper;
    MoveL Offs(pOrigin,93.18,51.54,0.00),v40,z0,tPen\WObj:=wPaper;
    MoveL Offs(pOrigin,93.18,49.41,0.00),v40,z0,tPen\WObj:=wPaper;
    MoveL Offs(pOrigin,93.88,46.44,0.00),v40,z0,tPen\WObj:=wPaper;
    MoveL Offs(pOrigin,94.88,44.95,0.00),v40,z0,tPen\WObj:=wPaper;
    MoveL Offs(pOrigin,96.79,43.04,0.00),v40,z0,tPen\WObj:=wPaper;
    MoveL Offs(pOrigin,98.49,41.90,0.00),v40,z0,tPen\WObj:=wPaper;
    MoveL Offs(pOrigin,101.68,40.49,0.00),v40,z0,tPen\WObj:=wPaper;
    MoveL Offs(pOrigin,105.71,39.64,0.00),v40,z0,tPen\WObj:=wPaper;
    MoveL Offs(pOrigin,108.05,39.64,0.00),v40,z0,tPen\WObj:=wPaper;
  ENDPROC

  PROC DrawPart50()
    MoveL Offs(pOrigin,108.19,40.06,0.00),v40,z0,tPen\WObj:=wPaper;
    MoveL Offs(pOrigin,107.77,41.12,0.00),v40,z0,tPen\WObj:=wPaper;
    MoveL Offs(pOrigin,106.07,43.46,0.00),v40,z0,tPen\WObj:=wPaper;
    MoveL Offs(pOrigin,105.07,47.50,0.00),v40,z0,tPen\WObj:=wPaper;
    MoveL Offs(pOrigin,105.71,52.17,0.00),v40,z0,tPen\WObj:=wPaper;
    MoveL Offs(pOrigin,106.99,55.58,0.00),v40,fine,tPen\WObj:=wPaper;
    MoveL Offs(pOrigin,106.99,55.58,6.00),v60,z5,tPen\WObj:=wPaper;
    MoveL Offs(pOrigin,96.57,58.34,6.00),vTravel,z5,tPen\WObj:=wPaper;
    MoveL Offs(pOrigin,96.57,58.34,0.00),v60,z0,tPen\WObj:=wPaper;
    MoveL Offs(pOrigin,96.79,58.76,0.00),v40,z0,tPen\WObj:=wPaper;
    MoveL Offs(pOrigin,96.57,58.34,0.00),v40,fine,tPen\WObj:=wPaper;
    MoveL Offs(pOrigin,96.57,58.34,6.00),v60,z5,tPen\WObj:=wPaper;
    MoveL Offs(pOrigin,95.94,61.95,6.00),vTravel,z5,tPen\WObj:=wPaper;
    MoveL Offs(pOrigin,95.94,61.95,0.00),v60,z0,tPen\WObj:=wPaper;
    MoveL Offs(pOrigin,96.15,62.38,0.00),v40,z0,tPen\WObj:=wPaper;
    MoveL Offs(pOrigin,95.94,61.95,0.00),v40,fine,tPen\WObj:=wPaper;
    MoveL Offs(pOrigin,95.94,61.95,6.00),v60,z5,tPen\WObj:=wPaper;
    MoveL Offs(pOrigin,98.91,63.22,6.00),vTravel,z5,tPen\WObj:=wPaper;
    MoveL Offs(pOrigin,98.91,63.22,0.00),v60,z0,tPen\WObj:=wPaper;
    MoveL Offs(pOrigin,99.12,63.65,0.00),v40,z0,tPen\WObj:=wPaper;
    MoveL Offs(pOrigin,98.91,63.22,0.00),v40,fine,tPen\WObj:=wPaper;
    MoveL Offs(pOrigin,98.91,63.22,6.00),v60,z5,tPen\WObj:=wPaper;
    MoveL Offs(pOrigin,100.61,64.71,6.00),vTravel,z5,tPen\WObj:=wPaper;
    MoveL Offs(pOrigin,100.61,64.71,0.00),v60,z0,tPen\WObj:=wPaper;
    MoveL Offs(pOrigin,102.10,66.20,0.00),v40,z0,tPen\WObj:=wPaper;
    MoveL Offs(pOrigin,100.61,64.71,0.00),v40,fine,tPen\WObj:=wPaper;
    MoveL Offs(pOrigin,100.61,64.71,6.00),v60,z5,tPen\WObj:=wPaper;
    MoveL Offs(pOrigin,92.75,67.26,6.00),vTravel,z5,tPen\WObj:=wPaper;
    MoveL Offs(pOrigin,92.75,67.26,0.00),v60,z0,tPen\WObj:=wPaper;
    MoveL Offs(pOrigin,94.38,70.45,0.00),v40,z0,tPen\WObj:=wPaper;
    MoveL Offs(pOrigin,96.36,73.21,0.00),v40,z0,tPen\WObj:=wPaper;
    MoveL Offs(pOrigin,100.40,77.25,0.00),v40,z0,tPen\WObj:=wPaper;
    MoveL Offs(pOrigin,106.35,81.93,0.00),v40,fine,tPen\WObj:=wPaper;
    MoveL Offs(pOrigin,106.35,81.93,6.00),v60,z5,tPen\WObj:=wPaper;
    MoveL Offs(pOrigin,104.44,80.65,6.00),vTravel,z5,tPen\WObj:=wPaper;
    MoveL Offs(pOrigin,104.44,80.65,0.00),v60,z0,tPen\WObj:=wPaper;
    MoveL Offs(pOrigin,105.07,81.07,0.00),v40,z0,tPen\WObj:=wPaper;
    MoveL Offs(pOrigin,104.44,80.65,0.00),v40,fine,tPen\WObj:=wPaper;
    MoveL Offs(pOrigin,104.44,80.65,6.00),v60,z5,tPen\WObj:=wPaper;
    MoveL Offs(pOrigin,108.90,80.44,6.00),vTravel,z5,tPen\WObj:=wPaper;
    MoveL Offs(pOrigin,108.90,80.44,0.00),v60,z0,tPen\WObj:=wPaper;
    MoveL Offs(pOrigin,109.96,81.50,0.00),v40,z0,tPen\WObj:=wPaper;
    MoveL Offs(pOrigin,108.90,80.44,0.00),v40,fine,tPen\WObj:=wPaper;
    MoveL Offs(pOrigin,108.90,80.44,6.00),v60,z5,tPen\WObj:=wPaper;
    MoveL Offs(pOrigin,112.09,77.04,6.00),vTravel,z5,tPen\WObj:=wPaper;
    MoveL Offs(pOrigin,112.09,77.04,0.00),v60,z0,tPen\WObj:=wPaper;
    MoveL Offs(pOrigin,112.51,77.46,0.00),v40,z0,tPen\WObj:=wPaper;
    MoveL Offs(pOrigin,112.09,77.04,0.00),v40,fine,tPen\WObj:=wPaper;
    MoveL Offs(pOrigin,112.09,77.04,6.00),v60,z5,tPen\WObj:=wPaper;
    MoveL Offs(pOrigin,110.60,75.34,6.00),vTravel,z5,tPen\WObj:=wPaper;
    MoveL Offs(pOrigin,110.60,75.34,0.00),v60,z0,tPen\WObj:=wPaper;
    MoveL Offs(pOrigin,111.03,75.76,0.00),v40,z0,tPen\WObj:=wPaper;
    MoveL Offs(pOrigin,110.60,75.34,0.00),v40,fine,tPen\WObj:=wPaper;
    MoveL Offs(pOrigin,110.60,75.34,6.00),v60,z5,tPen\WObj:=wPaper;
    MoveL Offs(pOrigin,114.64,74.91,6.00),vTravel,z5,tPen\WObj:=wPaper;
    MoveL Offs(pOrigin,114.64,74.91,0.00),v60,z0,tPen\WObj:=wPaper;
    MoveL Offs(pOrigin,120.16,79.02,0.00),v40,z0,tPen\WObj:=wPaper;
    MoveL Offs(pOrigin,123.56,80.93,0.00),v40,z0,tPen\WObj:=wPaper;
    MoveL Offs(pOrigin,127.60,82.42,0.00),v40,z0,tPen\WObj:=wPaper;
    MoveL Offs(pOrigin,128.24,83.41,0.00),v40,fine,tPen\WObj:=wPaper;
    MoveL Offs(pOrigin,128.24,83.41,6.00),v60,z5,tPen\WObj:=wPaper;
    MoveL Offs(pOrigin,116.55,90.43,6.00),vTravel,z5,tPen\WObj:=wPaper;
    MoveL Offs(pOrigin,116.55,90.43,0.00),v60,z0,tPen\WObj:=wPaper;
    MoveL Offs(pOrigin,110.81,88.37,0.00),v40,z0,tPen\WObj:=wPaper;
    MoveL Offs(pOrigin,105.29,85.40,0.00),v40,z0,tPen\WObj:=wPaper;
    MoveL Offs(pOrigin,100.40,81.71,0.00),v40,z0,tPen\WObj:=wPaper;
    MoveL Offs(pOrigin,97.28,78.74,0.00),v40,z0,tPen\WObj:=wPaper;
    MoveL Offs(pOrigin,96.36,77.46,0.00),v40,fine,tPen\WObj:=wPaper;
    MoveL Offs(pOrigin,96.36,77.46,6.00),v60,z5,tPen\WObj:=wPaper;
    MoveL Offs(pOrigin,96.79,73.85,6.00),vTravel,z5,tPen\WObj:=wPaper;
    MoveL Offs(pOrigin,96.79,73.85,0.00),v60,z0,tPen\WObj:=wPaper;
    MoveL Offs(pOrigin,98.70,75.76,0.00),v40,z0,tPen\WObj:=wPaper;
    MoveL Offs(pOrigin,96.79,73.85,0.00),v40,fine,tPen\WObj:=wPaper;
    MoveL Offs(pOrigin,96.79,73.85,6.00),v60,z5,tPen\WObj:=wPaper;
    MoveL Offs(pOrigin,95.72,82.35,6.00),vTravel,z5,tPen\WObj:=wPaper;
    MoveL Offs(pOrigin,95.72,82.35,0.00),v60,z0,tPen\WObj:=wPaper;
    MoveL Offs(pOrigin,95.94,82.78,0.00),v40,z0,tPen\WObj:=wPaper;
    MoveL Offs(pOrigin,95.72,82.35,0.00),v40,fine,tPen\WObj:=wPaper;
    MoveL Offs(pOrigin,95.72,82.35,6.00),v60,z5,tPen\WObj:=wPaper;
    MoveL Offs(pOrigin,127.60,60.67,6.00),vTravel,z5,tPen\WObj:=wPaper;
    MoveL Offs(pOrigin,127.60,60.67,0.00),v60,z0,tPen\WObj:=wPaper;
    MoveL Offs(pOrigin,125.83,56.85,0.00),v40,z0,tPen\WObj:=wPaper;
    MoveL Offs(pOrigin,124.41,51.75,0.00),v40,z0,tPen\WObj:=wPaper;
    MoveL Offs(pOrigin,124.41,47.50,0.00),v40,z0,tPen\WObj:=wPaper;
    MoveL Offs(pOrigin,125.62,43.89,0.00),v40,z0,tPen\WObj:=wPaper;
    MoveL Offs(pOrigin,127.46,41.55,0.00),v40,z0,tPen\WObj:=wPaper;
    MoveL Offs(pOrigin,127.74,40.49,0.00),v40,z0,tPen\WObj:=wPaper;
    MoveL Offs(pOrigin,127.18,39.92,0.00),v40,z0,tPen\WObj:=wPaper;
    MoveL Offs(pOrigin,123.99,39.78,0.00),v40,z0,tPen\WObj:=wPaper;
    MoveL Offs(pOrigin,122.71,41.76,0.00),v40,z0,tPen\WObj:=wPaper;
    MoveL Offs(pOrigin,121.08,42.83,0.00),v40,z0,tPen\WObj:=wPaper;
    MoveL Offs(pOrigin,120.16,46.86,0.00),v40,z0,tPen\WObj:=wPaper;
    MoveL Offs(pOrigin,120.16,49.84,0.00),v40,z0,tPen\WObj:=wPaper;
    MoveL Offs(pOrigin,120.80,52.39,0.00),v40,z0,tPen\WObj:=wPaper;
    MoveL Offs(pOrigin,120.80,52.39,0.00),v40,z0,tPen\WObj:=wPaper;
    MoveL Offs(pOrigin,121.86,53.03,0.00),v40,z0,tPen\WObj:=wPaper;
    MoveL Offs(pOrigin,123.70,56.42,0.00),v40,z0,tPen\WObj:=wPaper;
    MoveL Offs(pOrigin,126.54,60.46,0.00),v40,z0,tPen\WObj:=wPaper;
    MoveL Offs(pOrigin,127.81,61.31,0.00),v40,z0,tPen\WObj:=wPaper;
    MoveL Offs(pOrigin,130.57,64.50,0.00),v40,z0,tPen\WObj:=wPaper;
    MoveL Offs(pOrigin,131.00,65.99,0.00),v40,z0,tPen\WObj:=wPaper;
    MoveL Offs(pOrigin,131.00,65.99,0.00),v40,z0,tPen\WObj:=wPaper;
    MoveL Offs(pOrigin,129.73,65.70,0.00),v40,z0,tPen\WObj:=wPaper;
    MoveL Offs(pOrigin,126.11,63.44,0.00),v40,z0,tPen\WObj:=wPaper;
    MoveL Offs(pOrigin,123.14,60.67,0.00),v40,z0,tPen\WObj:=wPaper;
    MoveL Offs(pOrigin,121.79,58.34,0.00),v40,z0,tPen\WObj:=wPaper;
    MoveL Offs(pOrigin,121.22,56.64,0.00),v40,z0,tPen\WObj:=wPaper;
    MoveL Offs(pOrigin,120.59,53.03,0.00),v40,z0,tPen\WObj:=wPaper;
    MoveL Offs(pOrigin,120.80,52.39,0.00),v40,z0,tPen\WObj:=wPaper;
    MoveL Offs(pOrigin,120.59,51.96,0.00),v40,z0,tPen\WObj:=wPaper;
    MoveL Offs(pOrigin,120.80,52.39,0.00),v40,z0,tPen\WObj:=wPaper;
    MoveL Offs(pOrigin,120.59,51.96,0.00),v40,fine,tPen\WObj:=wPaper;
    MoveL Offs(pOrigin,120.59,51.96,6.00),v60,z5,tPen\WObj:=wPaper;
    MoveL Offs(pOrigin,122.50,53.88,6.00),vTravel,z5,tPen\WObj:=wPaper;
    MoveL Offs(pOrigin,122.50,53.88,0.00),v60,z0,tPen\WObj:=wPaper;
    MoveL Offs(pOrigin,122.71,54.30,0.00),v40,z0,tPen\WObj:=wPaper;
    MoveL Offs(pOrigin,122.50,53.88,0.00),v40,fine,tPen\WObj:=wPaper;
    MoveL Offs(pOrigin,122.50,53.88,6.00),v60,z5,tPen\WObj:=wPaper;
    MoveL Offs(pOrigin,126.54,58.12,6.00),vTravel,z5,tPen\WObj:=wPaper;
    MoveL Offs(pOrigin,126.54,58.12,0.00),v60,z0,tPen\WObj:=wPaper;
  ENDPROC

  PROC DrawPart51()
    MoveL Offs(pOrigin,126.75,58.55,0.00),v40,z0,tPen\WObj:=wPaper;
    MoveL Offs(pOrigin,126.54,58.12,0.00),v40,fine,tPen\WObj:=wPaper;
    MoveL Offs(pOrigin,126.54,58.12,6.00),v60,z5,tPen\WObj:=wPaper;
    MoveL Offs(pOrigin,131.00,65.99,6.00),vTravel,z5,tPen\WObj:=wPaper;
    MoveL Offs(pOrigin,131.00,65.99,0.00),v60,z0,tPen\WObj:=wPaper;
    MoveL Offs(pOrigin,135.25,68.61,0.00),v40,z0,tPen\WObj:=wPaper;
    MoveL Offs(pOrigin,142.48,71.80,0.00),v40,z0,tPen\WObj:=wPaper;
    MoveL Offs(pOrigin,147.36,73.43,0.00),v40,z0,tPen\WObj:=wPaper;
    MoveL Offs(pOrigin,152.46,74.49,0.00),v40,z0,tPen\WObj:=wPaper;
    MoveL Offs(pOrigin,154.80,74.70,0.00),v40,z0,tPen\WObj:=wPaper;
    MoveL Offs(pOrigin,157.99,74.49,0.00),v40,z0,tPen\WObj:=wPaper;
    MoveL Offs(pOrigin,162.66,73.43,0.00),v40,z0,tPen\WObj:=wPaper;
    MoveL Offs(pOrigin,166.70,71.58,0.00),v40,z0,tPen\WObj:=wPaper;
    MoveL Offs(pOrigin,167.69,70.88,0.00),v40,z0,tPen\WObj:=wPaper;
    MoveL Offs(pOrigin,168.19,70.03,0.00),v40,fine,tPen\WObj:=wPaper;
    MoveL Offs(pOrigin,168.19,70.03,6.00),v60,z5,tPen\WObj:=wPaper;
    MoveL Offs(pOrigin,167.12,68.96,6.00),vTravel,z5,tPen\WObj:=wPaper;
    MoveL Offs(pOrigin,167.12,68.96,0.00),v60,z0,tPen\WObj:=wPaper;
    MoveL Offs(pOrigin,165.00,68.82,0.00),v40,z0,tPen\WObj:=wPaper;
    MoveL Offs(pOrigin,163.09,69.18,0.00),v40,z0,tPen\WObj:=wPaper;
    MoveL Offs(pOrigin,163.09,69.18,0.00),v40,z0,tPen\WObj:=wPaper;
    MoveL Offs(pOrigin,162.45,68.75,0.00),v40,z0,tPen\WObj:=wPaper;
    MoveL Offs(pOrigin,157.77,68.96,0.00),v40,z0,tPen\WObj:=wPaper;
    MoveL Offs(pOrigin,157.77,68.96,0.00),v40,z0,tPen\WObj:=wPaper;
    MoveL Offs(pOrigin,157.14,68.25,0.00),v40,z0,tPen\WObj:=wPaper;
    MoveL Offs(pOrigin,154.16,67.12,0.00),v40,z0,tPen\WObj:=wPaper;
    MoveL Offs(pOrigin,150.98,64.93,0.00),v40,z0,tPen\WObj:=wPaper;
    MoveL Offs(pOrigin,147.57,61.31,0.00),v40,z0,tPen\WObj:=wPaper;
    MoveL Offs(pOrigin,146.02,58.97,0.00),v40,z0,tPen\WObj:=wPaper;
    MoveL Offs(pOrigin,144.32,55.79,0.00),v40,z0,tPen\WObj:=wPaper;
    MoveL Offs(pOrigin,142.48,50.47,0.00),v40,z0,tPen\WObj:=wPaper;
    MoveL Offs(pOrigin,142.90,45.59,0.00),v40,z0,tPen\WObj:=wPaper;
    MoveL Offs(pOrigin,143.11,44.74,0.00),v40,z0,tPen\WObj:=wPaper;
    MoveL Offs(pOrigin,142.90,45.16,0.00),v40,z0,tPen\WObj:=wPaper;
    MoveL Offs(pOrigin,143.11,44.74,0.00),v40,fine,tPen\WObj:=wPaper;
    MoveL Offs(pOrigin,143.11,44.74,6.00),v60,z5,tPen\WObj:=wPaper;
    MoveL Offs(pOrigin,145.45,42.19,6.00),vTravel,z5,tPen\WObj:=wPaper;
    MoveL Offs(pOrigin,145.45,42.19,0.00),v60,z0,tPen\WObj:=wPaper;
    MoveL Offs(pOrigin,145.88,41.97,0.00),v40,z0,tPen\WObj:=wPaper;
    MoveL Offs(pOrigin,145.45,42.19,0.00),v40,z0,tPen\WObj:=wPaper;
    MoveL Offs(pOrigin,146.30,41.76,0.00),v40,z0,tPen\WObj:=wPaper;
    MoveL Offs(pOrigin,146.73,41.55,0.00),v40,z0,tPen\WObj:=wPaper;
    MoveL Offs(pOrigin,146.30,41.76,0.00),v40,fine,tPen\WObj:=wPaper;
    MoveL Offs(pOrigin,146.30,41.76,6.00),v60,z5,tPen\WObj:=wPaper;
    MoveL Offs(pOrigin,143.32,40.91,6.00),vTravel,z5,tPen\WObj:=wPaper;
    MoveL Offs(pOrigin,143.32,40.91,0.00),v60,z0,tPen\WObj:=wPaper;
    MoveL Offs(pOrigin,143.96,40.35,0.00),v40,z0,tPen\WObj:=wPaper;
    MoveL Offs(pOrigin,146.73,39.21,0.00),v40,z0,tPen\WObj:=wPaper;
    MoveL Offs(pOrigin,149.70,39.00,0.00),v40,z0,tPen\WObj:=wPaper;
    MoveL Offs(pOrigin,150.34,39.64,0.00),v40,fine,tPen\WObj:=wPaper;
    MoveL Offs(pOrigin,150.34,39.64,6.00),v60,z5,tPen\WObj:=wPaper;
    MoveL Offs(pOrigin,154.38,37.51,6.00),vTravel,z5,tPen\WObj:=wPaper;
    MoveL Offs(pOrigin,154.38,37.51,0.00),v60,z0,tPen\WObj:=wPaper;
    MoveL Offs(pOrigin,153.74,37.09,0.00),v40,z0,tPen\WObj:=wPaper;
    MoveL Offs(pOrigin,149.49,36.45,0.00),v40,z0,tPen\WObj:=wPaper;
    MoveL Offs(pOrigin,145.45,36.45,0.00),v40,z0,tPen\WObj:=wPaper;
    MoveL Offs(pOrigin,142.90,36.88,0.00),v40,fine,tPen\WObj:=wPaper;
    MoveL Offs(pOrigin,142.90,36.88,6.00),v60,z5,tPen\WObj:=wPaper;
    MoveL Offs(pOrigin,140.56,39.42,6.00),vTravel,z5,tPen\WObj:=wPaper;
    MoveL Offs(pOrigin,140.56,39.42,0.00),v60,z0,tPen\WObj:=wPaper;
    MoveL Offs(pOrigin,140.35,39.85,0.00),v40,z0,tPen\WObj:=wPaper;
    MoveL Offs(pOrigin,140.56,39.42,0.00),v40,fine,tPen\WObj:=wPaper;
    MoveL Offs(pOrigin,140.56,39.42,6.00),v60,z5,tPen\WObj:=wPaper;
    MoveL Offs(pOrigin,142.90,41.12,6.00),vTravel,z5,tPen\WObj:=wPaper;
    MoveL Offs(pOrigin,142.90,41.12,0.00),v60,z0,tPen\WObj:=wPaper;
    MoveL Offs(pOrigin,140.77,43.46,0.00),v40,z0,tPen\WObj:=wPaper;
    MoveL Offs(pOrigin,139.71,45.80,0.00),v40,z0,tPen\WObj:=wPaper;
    MoveL Offs(pOrigin,139.71,45.80,0.00),v40,z0,tPen\WObj:=wPaper;
    MoveL Offs(pOrigin,138.86,45.94,0.00),v40,z0,tPen\WObj:=wPaper;
    MoveL Offs(pOrigin,138.37,46.44,0.00),v40,z0,tPen\WObj:=wPaper;
    MoveL Offs(pOrigin,137.38,48.78,0.00),v40,z0,tPen\WObj:=wPaper;
    MoveL Offs(pOrigin,137.16,50.26,0.00),v40,z0,tPen\WObj:=wPaper;
    MoveL Offs(pOrigin,137.16,50.26,0.00),v40,z0,tPen\WObj:=wPaper;
    MoveL Offs(pOrigin,138.01,50.69,0.00),v40,z0,tPen\WObj:=wPaper;
    MoveL Offs(pOrigin,138.65,51.54,0.00),v40,z0,tPen\WObj:=wPaper;
    MoveL Offs(pOrigin,138.65,51.54,0.00),v40,z0,tPen\WObj:=wPaper;
    MoveL Offs(pOrigin,139.29,51.54,0.00),v40,z0,tPen\WObj:=wPaper;
    MoveL Offs(pOrigin,140.14,52.81,0.00),v40,z0,tPen\WObj:=wPaper;
    MoveL Offs(pOrigin,140.14,53.24,0.00),v40,z0,tPen\WObj:=wPaper;
    MoveL Offs(pOrigin,140.56,52.81,0.00),v40,z0,tPen\WObj:=wPaper;
    MoveL Offs(pOrigin,141.55,53.03,0.00),v40,z0,tPen\WObj:=wPaper;
    MoveL Offs(pOrigin,142.83,56.64,0.00),v40,z0,tPen\WObj:=wPaper;
    MoveL Offs(pOrigin,144.53,59.83,0.00),v40,z0,tPen\WObj:=wPaper;
    MoveL Offs(pOrigin,146.51,62.59,0.00),v40,z0,tPen\WObj:=wPaper;
    MoveL Offs(pOrigin,148.21,64.29,0.00),v40,z0,tPen\WObj:=wPaper;
    MoveL Offs(pOrigin,148.21,64.29,0.00),v40,z0,tPen\WObj:=wPaper;
    MoveL Offs(pOrigin,148.64,64.50,0.00),v40,z0,tPen\WObj:=wPaper;
    MoveL Offs(pOrigin,148.64,64.93,0.00),v40,z0,tPen\WObj:=wPaper;
    MoveL Offs(pOrigin,148.64,64.93,0.00),v40,z0,tPen\WObj:=wPaper;
    MoveL Offs(pOrigin,149.06,64.93,0.00),v40,z0,tPen\WObj:=wPaper;
    MoveL Offs(pOrigin,150.12,65.78,0.00),v40,z0,tPen\WObj:=wPaper;
    MoveL Offs(pOrigin,149.91,66.41,0.00),v40,fine,tPen\WObj:=wPaper;
    MoveL Offs(pOrigin,149.91,66.41,6.00),v60,z5,tPen\WObj:=wPaper;
    MoveL Offs(pOrigin,152.46,66.20,6.00),vTravel,z5,tPen\WObj:=wPaper;
    MoveL Offs(pOrigin,152.46,66.20,0.00),v60,z0,tPen\WObj:=wPaper;
    MoveL Offs(pOrigin,152.89,66.41,0.00),v40,z0,tPen\WObj:=wPaper;
    MoveL Offs(pOrigin,152.46,66.20,0.00),v40,fine,tPen\WObj:=wPaper;
    MoveL Offs(pOrigin,152.46,66.20,6.00),v60,z5,tPen\WObj:=wPaper;
    MoveL Offs(pOrigin,153.52,68.96,6.00),vTravel,z5,tPen\WObj:=wPaper;
    MoveL Offs(pOrigin,153.52,68.96,0.00),v60,z0,tPen\WObj:=wPaper;
    MoveL Offs(pOrigin,147.79,65.14,0.00),v40,z0,tPen\WObj:=wPaper;
    MoveL Offs(pOrigin,144.60,62.16,0.00),v40,z0,tPen\WObj:=wPaper;
    MoveL Offs(pOrigin,144.60,62.16,0.00),v40,z0,tPen\WObj:=wPaper;
    MoveL Offs(pOrigin,144.39,62.59,0.00),v40,z0,tPen\WObj:=wPaper;
    MoveL Offs(pOrigin,144.81,62.38,0.00),v40,z0,tPen\WObj:=wPaper;
    MoveL Offs(pOrigin,143.96,61.95,0.00),v40,z0,tPen\WObj:=wPaper;
    MoveL Offs(pOrigin,144.60,64.71,0.00),v40,fine,tPen\WObj:=wPaper;
    MoveL Offs(pOrigin,144.60,64.71,6.00),v60,z5,tPen\WObj:=wPaper;
    MoveL Offs(pOrigin,145.88,65.78,6.00),vTravel,z5,tPen\WObj:=wPaper;
    MoveL Offs(pOrigin,145.88,65.78,0.00),v60,z0,tPen\WObj:=wPaper;
    MoveL Offs(pOrigin,146.30,66.20,0.00),v40,z0,tPen\WObj:=wPaper;
    MoveL Offs(pOrigin,145.88,65.78,0.00),v40,fine,tPen\WObj:=wPaper;
    MoveL Offs(pOrigin,145.88,65.78,6.00),v60,z5,tPen\WObj:=wPaper;
    MoveL Offs(pOrigin,146.09,63.44,6.00),vTravel,z5,tPen\WObj:=wPaper;
    MoveL Offs(pOrigin,146.09,63.44,0.00),v60,z0,tPen\WObj:=wPaper;
    MoveL Offs(pOrigin,146.94,64.29,0.00),v40,z0,tPen\WObj:=wPaper;
    MoveL Offs(pOrigin,146.09,63.44,0.00),v40,z0,tPen\WObj:=wPaper;
    MoveL Offs(pOrigin,146.51,62.38,0.00),v40,z0,tPen\WObj:=wPaper;
    MoveL Offs(pOrigin,147.15,63.01,0.00),v40,z0,tPen\WObj:=wPaper;
    MoveL Offs(pOrigin,146.51,62.38,0.00),v40,fine,tPen\WObj:=wPaper;
  ENDPROC

  PROC DrawPart52()
    MoveL Offs(pOrigin,146.51,62.38,6.00),v60,z5,tPen\WObj:=wPaper;
    MoveL Offs(pOrigin,143.96,61.95,6.00),vTravel,z5,tPen\WObj:=wPaper;
    MoveL Offs(pOrigin,143.96,61.95,0.00),v60,z0,tPen\WObj:=wPaper;
    MoveL Offs(pOrigin,142.90,60.89,0.00),v40,z0,tPen\WObj:=wPaper;
    MoveL Offs(pOrigin,142.90,60.89,0.00),v40,z0,tPen\WObj:=wPaper;
    MoveL Offs(pOrigin,141.84,60.25,0.00),v40,z0,tPen\WObj:=wPaper;
    MoveL Offs(pOrigin,141.84,59.61,0.00),v40,z0,tPen\WObj:=wPaper;
    MoveL Offs(pOrigin,142.48,59.40,0.00),v40,z0,tPen\WObj:=wPaper;
    MoveL Offs(pOrigin,142.26,59.61,0.00),v40,z0,tPen\WObj:=wPaper;
    MoveL Offs(pOrigin,141.84,59.40,0.00),v40,z0,tPen\WObj:=wPaper;
    MoveL Offs(pOrigin,142.26,58.97,0.00),v40,z0,tPen\WObj:=wPaper;
    MoveL Offs(pOrigin,142.05,58.34,0.00),v40,z0,tPen\WObj:=wPaper;
    MoveL Offs(pOrigin,143.32,60.25,0.00),v40,z0,tPen\WObj:=wPaper;
    MoveL Offs(pOrigin,143.11,60.25,0.00),v40,z0,tPen\WObj:=wPaper;
    MoveL Offs(pOrigin,143.11,60.25,0.00),v40,z0,tPen\WObj:=wPaper;
    MoveL Offs(pOrigin,143.32,60.67,0.00),v40,z0,tPen\WObj:=wPaper;
    MoveL Offs(pOrigin,142.90,60.46,0.00),v40,z0,tPen\WObj:=wPaper;
    MoveL Offs(pOrigin,143.11,60.25,0.00),v40,z0,tPen\WObj:=wPaper;
    MoveL Offs(pOrigin,143.32,60.67,0.00),v40,z0,tPen\WObj:=wPaper;
    MoveL Offs(pOrigin,142.90,60.46,0.00),v40,z0,tPen\WObj:=wPaper;
    MoveL Offs(pOrigin,143.11,60.25,0.00),v40,fine,tPen\WObj:=wPaper;
    MoveL Offs(pOrigin,143.11,60.25,6.00),v60,z5,tPen\WObj:=wPaper;
    MoveL Offs(pOrigin,141.62,58.76,6.00),vTravel,z5,tPen\WObj:=wPaper;
    MoveL Offs(pOrigin,141.62,58.76,0.00),v60,z0,tPen\WObj:=wPaper;
    MoveL Offs(pOrigin,140.77,58.34,0.00),v40,z0,tPen\WObj:=wPaper;
    MoveL Offs(pOrigin,140.56,57.06,0.00),v40,z0,tPen\WObj:=wPaper;
    MoveL Offs(pOrigin,140.35,56.42,0.00),v40,z0,tPen\WObj:=wPaper;
    MoveL Offs(pOrigin,140.77,56.00,0.00),v40,z0,tPen\WObj:=wPaper;
    MoveL Offs(pOrigin,140.99,56.42,0.00),v40,z0,tPen\WObj:=wPaper;
    MoveL Offs(pOrigin,140.99,56.42,0.00),v40,z0,tPen\WObj:=wPaper;
    MoveL Offs(pOrigin,141.84,57.49,0.00),v40,z0,tPen\WObj:=wPaper;
    MoveL Offs(pOrigin,142.05,58.34,0.00),v40,fine,tPen\WObj:=wPaper;
    MoveL Offs(pOrigin,142.05,58.34,6.00),v60,z5,tPen\WObj:=wPaper;
    MoveL Offs(pOrigin,140.35,56.42,6.00),vTravel,z5,tPen\WObj:=wPaper;
    MoveL Offs(pOrigin,140.35,56.42,0.00),v60,z0,tPen\WObj:=wPaper;
    MoveL Offs(pOrigin,139.93,56.21,0.00),v40,z0,tPen\WObj:=wPaper;
    MoveL Offs(pOrigin,139.93,55.79,0.00),v40,z0,tPen\WObj:=wPaper;
    MoveL Offs(pOrigin,140.77,55.58,0.00),v40,z0,tPen\WObj:=wPaper;
    MoveL Offs(pOrigin,140.56,54.72,0.00),v40,z0,tPen\WObj:=wPaper;
    MoveL Offs(pOrigin,139.71,54.94,0.00),v40,z0,tPen\WObj:=wPaper;
    MoveL Offs(pOrigin,139.29,54.51,0.00),v40,z0,tPen\WObj:=wPaper;
    MoveL Offs(pOrigin,140.35,54.09,0.00),v40,z0,tPen\WObj:=wPaper;
    MoveL Offs(pOrigin,140.14,53.24,0.00),v40,z0,tPen\WObj:=wPaper;
    MoveL Offs(pOrigin,139.07,53.45,0.00),v40,z0,tPen\WObj:=wPaper;
    MoveL Offs(pOrigin,139.07,53.45,0.00),v40,z0,tPen\WObj:=wPaper;
    MoveL Offs(pOrigin,138.44,52.81,0.00),v40,z0,tPen\WObj:=wPaper;
    MoveL Offs(pOrigin,138.65,51.54,0.00),v40,z0,tPen\WObj:=wPaper;
    MoveL Offs(pOrigin,138.65,51.54,0.00),v40,z0,tPen\WObj:=wPaper;
    MoveL Offs(pOrigin,138.01,50.90,0.00),v40,z0,tPen\WObj:=wPaper;
    MoveL Offs(pOrigin,137.16,50.26,0.00),v40,z0,tPen\WObj:=wPaper;
    MoveL Offs(pOrigin,136.52,51.33,0.00),v40,z0,tPen\WObj:=wPaper;
    MoveL Offs(pOrigin,136.52,54.72,0.00),v40,z0,tPen\WObj:=wPaper;
    MoveL Offs(pOrigin,137.94,58.55,0.00),v40,z0,tPen\WObj:=wPaper;
    MoveL Offs(pOrigin,139.93,61.31,0.00),v40,z0,tPen\WObj:=wPaper;
    MoveL Offs(pOrigin,142.90,64.22,0.00),v40,z0,tPen\WObj:=wPaper;
    MoveL Offs(pOrigin,144.60,64.85,0.00),v40,z0,tPen\WObj:=wPaper;
    MoveL Offs(pOrigin,146.94,66.84,0.00),v40,z0,tPen\WObj:=wPaper;
    MoveL Offs(pOrigin,152.04,69.88,0.00),v40,z0,tPen\WObj:=wPaper;
    MoveL Offs(pOrigin,153.10,70.03,0.00),v40,z0,tPen\WObj:=wPaper;
    MoveL Offs(pOrigin,153.10,70.03,0.00),v40,z0,tPen\WObj:=wPaper;
    MoveL Offs(pOrigin,153.31,70.38,0.00),v40,z0,tPen\WObj:=wPaper;
    MoveL Offs(pOrigin,155.44,71.09,0.00),v40,z0,tPen\WObj:=wPaper;
    MoveL Offs(pOrigin,159.69,71.30,0.00),v40,z0,tPen\WObj:=wPaper;
    MoveL Offs(pOrigin,162.59,70.38,0.00),v40,z0,tPen\WObj:=wPaper;
    MoveL Offs(pOrigin,163.09,69.18,0.00),v40,fine,tPen\WObj:=wPaper;
    MoveL Offs(pOrigin,163.09,69.18,6.00),v60,z5,tPen\WObj:=wPaper;
    MoveL Offs(pOrigin,163.51,65.35,6.00),vTravel,z5,tPen\WObj:=wPaper;
    MoveL Offs(pOrigin,163.51,65.35,0.00),v60,z0,tPen\WObj:=wPaper;
    MoveL Offs(pOrigin,166.49,67.47,0.00),v40,z0,tPen\WObj:=wPaper;
    MoveL Offs(pOrigin,167.12,68.96,0.00),v40,z0,tPen\WObj:=wPaper;
    MoveL Offs(pOrigin,167.12,68.96,0.00),v40,z0,tPen\WObj:=wPaper;
    MoveL Offs(pOrigin,167.90,69.25,0.00),v40,z0,tPen\WObj:=wPaper;
    MoveL Offs(pOrigin,168.40,69.95,0.00),v40,z0,tPen\WObj:=wPaper;
    MoveL Offs(pOrigin,169.89,70.45,0.00),v40,z0,tPen\WObj:=wPaper;
    MoveL Offs(pOrigin,170.60,71.30,0.00),v40,z0,tPen\WObj:=wPaper;
    MoveL Offs(pOrigin,170.74,72.15,0.00),v40,z0,tPen\WObj:=wPaper;
    MoveL Offs(pOrigin,170.74,72.15,0.00),v40,z0,tPen\WObj:=wPaper;
    MoveL Offs(pOrigin,169.04,73.43,0.00),v40,fine,tPen\WObj:=wPaper;
    MoveL Offs(pOrigin,169.04,73.43,6.00),v60,z5,tPen\WObj:=wPaper;
    MoveL Offs(pOrigin,170.74,72.15,6.00),vTravel,z5,tPen\WObj:=wPaper;
    MoveL Offs(pOrigin,170.74,72.15,0.00),v60,z0,tPen\WObj:=wPaper;
    MoveL Offs(pOrigin,172.01,72.57,0.00),v40,z0,tPen\WObj:=wPaper;
    MoveL Offs(pOrigin,176.69,76.68,0.00),v40,z0,tPen\WObj:=wPaper;
    MoveL Offs(pOrigin,179.24,77.68,0.00),v40,z0,tPen\WObj:=wPaper;
    MoveL Offs(pOrigin,181.36,77.89,0.00),v40,fine,tPen\WObj:=wPaper;
    MoveL Offs(pOrigin,181.36,77.89,6.00),v60,z5,tPen\WObj:=wPaper;
    MoveL Offs(pOrigin,180.51,82.99,6.00),vTravel,z5,tPen\WObj:=wPaper;
    MoveL Offs(pOrigin,180.51,82.99,0.00),v60,z0,tPen\WObj:=wPaper;
    MoveL Offs(pOrigin,180.30,83.41,0.00),v40,z0,tPen\WObj:=wPaper;
    MoveL Offs(pOrigin,180.51,82.99,0.00),v40,fine,tPen\WObj:=wPaper;
    MoveL Offs(pOrigin,180.51,82.99,6.00),v60,z5,tPen\WObj:=wPaper;
    MoveL Offs(pOrigin,181.15,85.96,6.00),vTravel,z5,tPen\WObj:=wPaper;
    MoveL Offs(pOrigin,181.15,85.96,0.00),v60,z0,tPen\WObj:=wPaper;
    MoveL Offs(pOrigin,180.73,86.39,0.00),v40,z0,tPen\WObj:=wPaper;
    MoveL Offs(pOrigin,181.15,85.96,0.00),v40,fine,tPen\WObj:=wPaper;
    MoveL Offs(pOrigin,181.15,85.96,6.00),v60,z5,tPen\WObj:=wPaper;
    MoveL Offs(pOrigin,179.45,87.45,6.00),vTravel,z5,tPen\WObj:=wPaper;
    MoveL Offs(pOrigin,179.45,87.45,0.00),v60,z0,tPen\WObj:=wPaper;
    MoveL Offs(pOrigin,179.02,87.88,0.00),v40,z0,tPen\WObj:=wPaper;
    MoveL Offs(pOrigin,179.45,87.45,0.00),v40,fine,tPen\WObj:=wPaper;
    MoveL Offs(pOrigin,179.45,87.45,6.00),v60,z5,tPen\WObj:=wPaper;
    MoveL Offs(pOrigin,180.09,89.36,6.00),vTravel,z5,tPen\WObj:=wPaper;
    MoveL Offs(pOrigin,180.09,89.36,0.00),v60,z0,tPen\WObj:=wPaper;
    MoveL Offs(pOrigin,179.66,89.79,0.00),v40,z0,tPen\WObj:=wPaper;
    MoveL Offs(pOrigin,180.09,89.36,0.00),v40,fine,tPen\WObj:=wPaper;
    MoveL Offs(pOrigin,180.09,89.36,6.00),v60,z5,tPen\WObj:=wPaper;
    MoveL Offs(pOrigin,184.12,86.18,6.00),vTravel,z5,tPen\WObj:=wPaper;
    MoveL Offs(pOrigin,184.12,86.18,0.00),v60,z0,tPen\WObj:=wPaper;
    MoveL Offs(pOrigin,184.34,85.75,0.00),v40,z0,tPen\WObj:=wPaper;
    MoveL Offs(pOrigin,184.12,86.18,0.00),v40,fine,tPen\WObj:=wPaper;
    MoveL Offs(pOrigin,184.12,86.18,6.00),v60,z5,tPen\WObj:=wPaper;
    MoveL Offs(pOrigin,176.26,83.20,6.00),vTravel,z5,tPen\WObj:=wPaper;
    MoveL Offs(pOrigin,176.26,83.20,0.00),v60,z0,tPen\WObj:=wPaper;
    MoveL Offs(pOrigin,175.62,83.84,0.00),v40,z0,tPen\WObj:=wPaper;
    MoveL Offs(pOrigin,176.26,83.20,0.00),v40,fine,tPen\WObj:=wPaper;
    MoveL Offs(pOrigin,176.26,83.20,6.00),v60,z5,tPen\WObj:=wPaper;
    MoveL Offs(pOrigin,174.99,84.26,6.00),vTravel,z5,tPen\WObj:=wPaper;
    MoveL Offs(pOrigin,174.99,84.26,0.00),v60,z0,tPen\WObj:=wPaper;
    MoveL Offs(pOrigin,173.93,85.32,0.00),v40,z0,tPen\WObj:=wPaper;
    MoveL Offs(pOrigin,174.99,84.26,0.00),v40,fine,tPen\WObj:=wPaper;
  ENDPROC

  PROC DrawPart53()
    MoveL Offs(pOrigin,174.99,84.26,6.00),v60,z5,tPen\WObj:=wPaper;
    MoveL Offs(pOrigin,172.01,87.03,6.00),vTravel,z5,tPen\WObj:=wPaper;
    MoveL Offs(pOrigin,172.01,87.03,0.00),v60,z0,tPen\WObj:=wPaper;
    MoveL Offs(pOrigin,171.59,87.45,0.00),v40,z0,tPen\WObj:=wPaper;
    MoveL Offs(pOrigin,172.01,87.03,0.00),v40,fine,tPen\WObj:=wPaper;
    MoveL Offs(pOrigin,172.01,87.03,6.00),v60,z5,tPen\WObj:=wPaper;
    MoveL Offs(pOrigin,167.98,76.61,6.00),vTravel,z5,tPen\WObj:=wPaper;
    MoveL Offs(pOrigin,167.98,76.61,0.00),v60,z0,tPen\WObj:=wPaper;
    MoveL Offs(pOrigin,167.76,77.04,0.00),v40,z0,tPen\WObj:=wPaper;
    MoveL Offs(pOrigin,167.98,76.61,0.00),v40,z0,tPen\WObj:=wPaper;
    MoveL Offs(pOrigin,168.40,75.76,0.00),v40,z0,tPen\WObj:=wPaper;
    MoveL Offs(pOrigin,168.19,76.19,0.00),v40,z0,tPen\WObj:=wPaper;
    MoveL Offs(pOrigin,168.40,75.76,0.00),v40,fine,tPen\WObj:=wPaper;
    MoveL Offs(pOrigin,168.40,75.76,6.00),v60,z5,tPen\WObj:=wPaper;
    MoveL Offs(pOrigin,172.44,72.79,6.00),vTravel,z5,tPen\WObj:=wPaper;
    MoveL Offs(pOrigin,172.44,72.79,0.00),v60,z0,tPen\WObj:=wPaper;
    MoveL Offs(pOrigin,174.14,74.49,0.00),v40,z0,tPen\WObj:=wPaper;
    MoveL Offs(pOrigin,172.44,72.79,0.00),v40,fine,tPen\WObj:=wPaper;
    MoveL Offs(pOrigin,172.44,72.79,6.00),v60,z5,tPen\WObj:=wPaper;
    MoveL Offs(pOrigin,163.30,64.07,6.00),vTravel,z5,tPen\WObj:=wPaper;
    MoveL Offs(pOrigin,163.30,64.07,0.00),v60,z0,tPen\WObj:=wPaper;
    MoveL Offs(pOrigin,161.18,60.67,0.00),v40,fine,tPen\WObj:=wPaper;
    MoveL Offs(pOrigin,161.18,60.67,6.00),v60,z5,tPen\WObj:=wPaper;
    MoveL Offs(pOrigin,157.77,68.96,6.00),vTravel,z5,tPen\WObj:=wPaper;
    MoveL Offs(pOrigin,157.77,68.96,0.00),v60,z0,tPen\WObj:=wPaper;
    MoveL Offs(pOrigin,156.93,69.60,0.00),v40,z0,tPen\WObj:=wPaper;
    MoveL Offs(pOrigin,153.52,68.96,0.00),v40,z0,tPen\WObj:=wPaper;
    MoveL Offs(pOrigin,153.52,68.96,0.00),v40,z0,tPen\WObj:=wPaper;
    MoveL Offs(pOrigin,153.10,70.03,0.00),v40,fine,tPen\WObj:=wPaper;
    MoveL Offs(pOrigin,153.10,70.03,6.00),v60,z5,tPen\WObj:=wPaper;
    MoveL Offs(pOrigin,152.68,80.86,6.00),vTravel,z5,tPen\WObj:=wPaper;
    MoveL Offs(pOrigin,152.68,80.86,0.00),v60,z0,tPen\WObj:=wPaper;
    MoveL Offs(pOrigin,150.48,83.41,0.00),v40,z0,tPen\WObj:=wPaper;
    MoveL Offs(pOrigin,144.60,88.94,0.00),v40,fine,tPen\WObj:=wPaper;
    MoveL Offs(pOrigin,144.60,88.94,6.00),v60,z5,tPen\WObj:=wPaper;
    MoveL Offs(pOrigin,146.51,87.24,6.00),vTravel,z5,tPen\WObj:=wPaper;
    MoveL Offs(pOrigin,146.51,87.24,0.00),v60,z0,tPen\WObj:=wPaper;
    MoveL Offs(pOrigin,146.30,87.66,0.00),v40,z0,tPen\WObj:=wPaper;
    MoveL Offs(pOrigin,146.51,87.24,0.00),v40,z0,tPen\WObj:=wPaper;
    MoveL Offs(pOrigin,146.94,87.03,0.00),v40,z0,tPen\WObj:=wPaper;
    MoveL Offs(pOrigin,147.15,86.60,0.00),v40,z0,tPen\WObj:=wPaper;
    MoveL Offs(pOrigin,146.94,87.03,0.00),v40,fine,tPen\WObj:=wPaper;
    MoveL Offs(pOrigin,146.94,87.03,6.00),v60,z5,tPen\WObj:=wPaper;
    MoveL Offs(pOrigin,147.79,85.96,6.00),vTravel,z5,tPen\WObj:=wPaper;
    MoveL Offs(pOrigin,147.79,85.96,0.00),v60,z0,tPen\WObj:=wPaper;
    MoveL Offs(pOrigin,147.57,86.39,0.00),v40,z0,tPen\WObj:=wPaper;
    MoveL Offs(pOrigin,147.79,85.96,0.00),v40,z0,tPen\WObj:=wPaper;
    MoveL Offs(pOrigin,148.21,85.75,0.00),v40,z0,tPen\WObj:=wPaper;
    MoveL Offs(pOrigin,148.43,85.32,0.00),v40,z0,tPen\WObj:=wPaper;
    MoveL Offs(pOrigin,148.21,85.75,0.00),v40,fine,tPen\WObj:=wPaper;
    MoveL Offs(pOrigin,148.21,85.75,6.00),v60,z5,tPen\WObj:=wPaper;
    MoveL Offs(pOrigin,149.06,84.69,6.00),vTravel,z5,tPen\WObj:=wPaper;
    MoveL Offs(pOrigin,149.06,84.69,0.00),v60,z0,tPen\WObj:=wPaper;
    MoveL Offs(pOrigin,148.85,85.11,0.00),v40,z0,tPen\WObj:=wPaper;
    MoveL Offs(pOrigin,149.06,84.69,0.00),v40,z0,tPen\WObj:=wPaper;
    MoveL Offs(pOrigin,149.49,84.47,0.00),v40,z0,tPen\WObj:=wPaper;
    MoveL Offs(pOrigin,149.70,84.05,0.00),v40,z0,tPen\WObj:=wPaper;
    MoveL Offs(pOrigin,149.49,84.47,0.00),v40,z0,tPen\WObj:=wPaper;
    MoveL Offs(pOrigin,150.12,83.84,0.00),v40,z0,tPen\WObj:=wPaper;
    MoveL Offs(pOrigin,150.34,83.41,0.00),v40,z0,tPen\WObj:=wPaper;
    MoveL Offs(pOrigin,150.12,83.84,0.00),v40,fine,tPen\WObj:=wPaper;
    MoveL Offs(pOrigin,150.12,83.84,6.00),v60,z5,tPen\WObj:=wPaper;
    MoveL Offs(pOrigin,152.04,86.81,6.00),vTravel,z5,tPen\WObj:=wPaper;
    MoveL Offs(pOrigin,152.04,86.81,0.00),v60,z0,tPen\WObj:=wPaper;
    MoveL Offs(pOrigin,150.55,88.30,0.00),v40,z0,tPen\WObj:=wPaper;
    MoveL Offs(pOrigin,152.04,86.81,0.00),v40,fine,tPen\WObj:=wPaper;
    MoveL Offs(pOrigin,152.04,86.81,6.00),v60,z5,tPen\WObj:=wPaper;
    MoveL Offs(pOrigin,153.52,85.11,6.00),vTravel,z5,tPen\WObj:=wPaper;
    MoveL Offs(pOrigin,153.52,85.11,0.00),v60,z0,tPen\WObj:=wPaper;
    MoveL Offs(pOrigin,152.68,85.96,0.00),v40,z0,tPen\WObj:=wPaper;
    MoveL Offs(pOrigin,153.52,85.11,0.00),v40,fine,tPen\WObj:=wPaper;
    MoveL Offs(pOrigin,153.52,85.11,6.00),v60,z5,tPen\WObj:=wPaper;
    MoveL Offs(pOrigin,142.48,63.65,6.00),vTravel,z5,tPen\WObj:=wPaper;
    MoveL Offs(pOrigin,142.48,63.65,0.00),v60,z0,tPen\WObj:=wPaper;
    MoveL Offs(pOrigin,142.90,64.07,0.00),v40,z0,tPen\WObj:=wPaper;
    MoveL Offs(pOrigin,142.48,63.65,0.00),v40,fine,tPen\WObj:=wPaper;
    MoveL Offs(pOrigin,142.48,63.65,6.00),v60,z5,tPen\WObj:=wPaper;
    MoveL Offs(pOrigin,141.41,62.59,6.00),vTravel,z5,tPen\WObj:=wPaper;
    MoveL Offs(pOrigin,141.41,62.59,0.00),v60,z0,tPen\WObj:=wPaper;
    MoveL Offs(pOrigin,142.26,63.44,0.00),v40,z0,tPen\WObj:=wPaper;
    MoveL Offs(pOrigin,141.41,62.59,0.00),v40,z0,tPen\WObj:=wPaper;
    MoveL Offs(pOrigin,140.77,61.95,0.00),v40,z0,tPen\WObj:=wPaper;
    MoveL Offs(pOrigin,141.20,62.38,0.00),v40,z0,tPen\WObj:=wPaper;
    MoveL Offs(pOrigin,140.77,61.95,0.00),v40,fine,tPen\WObj:=wPaper;
    MoveL Offs(pOrigin,140.77,61.95,6.00),v60,z5,tPen\WObj:=wPaper;
    MoveL Offs(pOrigin,137.80,57.91,6.00),vTravel,z5,tPen\WObj:=wPaper;
    MoveL Offs(pOrigin,137.80,57.91,0.00),v60,z0,tPen\WObj:=wPaper;
    MoveL Offs(pOrigin,138.01,58.34,0.00),v40,z0,tPen\WObj:=wPaper;
    MoveL Offs(pOrigin,137.80,57.91,0.00),v40,fine,tPen\WObj:=wPaper;
    MoveL Offs(pOrigin,137.80,57.91,6.00),v60,z5,tPen\WObj:=wPaper;
    MoveL Offs(pOrigin,144.60,56.64,6.00),vTravel,z5,tPen\WObj:=wPaper;
    MoveL Offs(pOrigin,144.60,56.64,0.00),v60,z0,tPen\WObj:=wPaper;
    MoveL Offs(pOrigin,144.81,57.06,0.00),v40,z0,tPen\WObj:=wPaper;
    MoveL Offs(pOrigin,144.60,56.64,0.00),v40,fine,tPen\WObj:=wPaper;
    MoveL Offs(pOrigin,144.60,56.64,6.00),v60,z5,tPen\WObj:=wPaper;
    MoveL Offs(pOrigin,142.90,52.60,6.00),vTravel,z5,tPen\WObj:=wPaper;
    MoveL Offs(pOrigin,142.90,52.60,0.00),v60,z0,tPen\WObj:=wPaper;
    MoveL Offs(pOrigin,141.62,52.60,0.00),v40,z0,tPen\WObj:=wPaper;
    MoveL Offs(pOrigin,141.20,52.17,0.00),v40,z0,tPen\WObj:=wPaper;
    MoveL Offs(pOrigin,141.27,51.11,0.00),v40,z0,tPen\WObj:=wPaper;
    MoveL Offs(pOrigin,142.48,50.90,0.00),v40,fine,tPen\WObj:=wPaper;
    MoveL Offs(pOrigin,142.48,50.90,6.00),v60,z5,tPen\WObj:=wPaper;
    MoveL Offs(pOrigin,138.23,42.40,6.00),vTravel,z5,tPen\WObj:=wPaper;
    MoveL Offs(pOrigin,138.23,42.40,0.00),v60,z0,tPen\WObj:=wPaper;
    MoveL Offs(pOrigin,138.01,42.83,0.00),v40,z0,tPen\WObj:=wPaper;
    MoveL Offs(pOrigin,138.23,42.40,0.00),v40,fine,tPen\WObj:=wPaper;
    MoveL Offs(pOrigin,138.23,42.40,6.00),v60,z5,tPen\WObj:=wPaper;
    MoveL Offs(pOrigin,131.43,38.58,6.00),vTravel,z5,tPen\WObj:=wPaper;
    MoveL Offs(pOrigin,131.43,38.58,0.00),v60,z0,tPen\WObj:=wPaper;
    MoveL Offs(pOrigin,130.57,37.80,0.00),v40,z0,tPen\WObj:=wPaper;
    MoveL Offs(pOrigin,108.90,35.39,0.00),v40,z0,tPen\WObj:=wPaper;
    MoveL Offs(pOrigin,98.91,33.90,0.00),v40,fine,tPen\WObj:=wPaper;
    MoveL Offs(pOrigin,98.91,33.90,6.00),v60,z5,tPen\WObj:=wPaper;
    MoveL Offs(pOrigin,96.15,43.46,6.00),vTravel,z5,tPen\WObj:=wPaper;
    MoveL Offs(pOrigin,96.15,43.46,0.00),v60,z0,tPen\WObj:=wPaper;
    MoveL Offs(pOrigin,95.30,44.31,0.00),v40,z0,tPen\WObj:=wPaper;
    MoveL Offs(pOrigin,96.15,43.46,0.00),v40,fine,tPen\WObj:=wPaper;
    MoveL Offs(pOrigin,96.15,43.46,6.00),v60,z5,tPen\WObj:=wPaper;
    MoveL Offs(pOrigin,106.56,42.40,6.00),vTravel,z5,tPen\WObj:=wPaper;
    MoveL Offs(pOrigin,106.56,42.40,0.00),v60,z0,tPen\WObj:=wPaper;
  ENDPROC

  PROC DrawPart54()
    MoveL Offs(pOrigin,106.35,42.83,0.00),v40,z0,tPen\WObj:=wPaper;
    MoveL Offs(pOrigin,106.56,42.40,0.00),v40,fine,tPen\WObj:=wPaper;
    MoveL Offs(pOrigin,106.56,42.40,6.00),v60,z5,tPen\WObj:=wPaper;
    MoveL Offs(pOrigin,107.62,41.12,6.00),vTravel,z5,tPen\WObj:=wPaper;
    MoveL Offs(pOrigin,107.62,41.12,0.00),v60,z0,tPen\WObj:=wPaper;
    MoveL Offs(pOrigin,107.41,41.55,0.00),v40,z0,tPen\WObj:=wPaper;
    MoveL Offs(pOrigin,107.62,41.12,0.00),v40,fine,tPen\WObj:=wPaper;
    MoveL Offs(pOrigin,107.62,41.12,6.00),v60,z5,tPen\WObj:=wPaper;
    MoveL Offs(pOrigin,112.51,40.70,6.00),vTravel,z5,tPen\WObj:=wPaper;
    MoveL Offs(pOrigin,112.51,40.70,0.00),v60,z0,tPen\WObj:=wPaper;
    MoveL Offs(pOrigin,111.52,41.20,0.00),v40,z0,tPen\WObj:=wPaper;
    MoveL Offs(pOrigin,110.60,43.46,0.00),v40,z0,tPen\WObj:=wPaper;
    MoveL Offs(pOrigin,110.81,44.74,0.00),v40,z0,tPen\WObj:=wPaper;
    MoveL Offs(pOrigin,111.24,44.95,0.00),v40,z0,tPen\WObj:=wPaper;
    MoveL Offs(pOrigin,112.30,44.74,0.00),v40,fine,tPen\WObj:=wPaper;
    MoveL Offs(pOrigin,112.30,44.74,6.00),v60,z5,tPen\WObj:=wPaper;
    MoveL Offs(pOrigin,114.21,44.10,6.00),vTravel,z5,tPen\WObj:=wPaper;
    MoveL Offs(pOrigin,114.21,44.10,0.00),v60,z0,tPen\WObj:=wPaper;
    MoveL Offs(pOrigin,114.43,41.97,0.00),v40,z0,tPen\WObj:=wPaper;
    MoveL Offs(pOrigin,115.35,39.00,0.00),v40,z0,tPen\WObj:=wPaper;
    MoveL Offs(pOrigin,115.70,38.79,0.00),v40,z0,tPen\WObj:=wPaper;
    MoveL Offs(pOrigin,117.82,39.00,0.00),v40,fine,tPen\WObj:=wPaper;
    MoveL Offs(pOrigin,117.82,39.00,6.00),v60,z5,tPen\WObj:=wPaper;
    MoveL Offs(pOrigin,115.28,38.79,6.00),vTravel,z5,tPen\WObj:=wPaper;
    MoveL Offs(pOrigin,115.28,38.79,0.00),v60,z0,tPen\WObj:=wPaper;
    MoveL Offs(pOrigin,114.64,38.58,0.00),v40,z0,tPen\WObj:=wPaper;
    MoveL Offs(pOrigin,113.15,38.79,0.00),v40,fine,tPen\WObj:=wPaper;
    MoveL Offs(pOrigin,113.15,38.79,6.00),v60,z5,tPen\WObj:=wPaper;
    MoveL Offs(pOrigin,130.79,37.72,6.00),vTravel,z5,tPen\WObj:=wPaper;
    MoveL Offs(pOrigin,130.79,37.72,0.00),v60,z0,tPen\WObj:=wPaper;
    MoveL Offs(pOrigin,131.43,38.58,0.00),v40,fine,tPen\WObj:=wPaper;
    MoveL Offs(pOrigin,131.43,38.58,6.00),v60,z5,tPen\WObj:=wPaper;
    MoveL Offs(pOrigin,88.07,32.41,6.00),vTravel,z5,tPen\WObj:=wPaper;
    MoveL Offs(pOrigin,88.07,32.41,0.00),v60,z0,tPen\WObj:=wPaper;
    MoveL Offs(pOrigin,88.71,31.99,0.00),v40,z0,tPen\WObj:=wPaper;
    MoveL Offs(pOrigin,186.68,22.85,0.00),v40,z0,tPen\WObj:=wPaper;
    MoveL Offs(pOrigin,192.62,22.21,0.00),v40,z0,tPen\WObj:=wPaper;
    MoveL Offs(pOrigin,194.54,21.58,0.00),v40,fine,tPen\WObj:=wPaper;
    MoveL Offs(pOrigin,194.54,21.58,6.00),v60,z5,tPen\WObj:=wPaper;
    MoveL Offs(pOrigin,196.66,20.73,6.00),vTravel,z5,tPen\WObj:=wPaper;
    MoveL Offs(pOrigin,196.66,20.73,0.00),v60,z0,tPen\WObj:=wPaper;
    MoveL Offs(pOrigin,195.81,19.02,0.00),v40,z0,tPen\WObj:=wPaper;
    MoveL Offs(pOrigin,195.81,17.11,0.00),v40,fine,tPen\WObj:=wPaper;
    MoveL Offs(pOrigin,195.81,17.11,6.00),v60,z5,tPen\WObj:=wPaper;
    MoveL Offs(pOrigin,199.43,33.69,6.00),vTravel,z5,tPen\WObj:=wPaper;
    MoveL Offs(pOrigin,199.43,33.69,0.00),v60,z0,tPen\WObj:=wPaper;
    MoveL Offs(pOrigin,200.27,34.75,0.00),v40,z0,tPen\WObj:=wPaper;
    MoveL Offs(pOrigin,200.70,36.03,0.00),v40,z0,tPen\WObj:=wPaper;
    MoveL Offs(pOrigin,200.70,36.03,0.00),v40,z0,tPen\WObj:=wPaper;
    MoveL Offs(pOrigin,200.06,36.45,0.00),v40,z0,tPen\WObj:=wPaper;
    MoveL Offs(pOrigin,199.21,36.24,0.00),v40,z0,tPen\WObj:=wPaper;
    MoveL Offs(pOrigin,194.11,36.45,0.00),v40,z0,tPen\WObj:=wPaper;
    MoveL Offs(pOrigin,189.23,37.94,0.00),v40,z0,tPen\WObj:=wPaper;
    MoveL Offs(pOrigin,189.23,37.94,0.00),v40,z0,tPen\WObj:=wPaper;
    MoveL Offs(pOrigin,190.71,39.42,0.00),v40,z0,tPen\WObj:=wPaper;
    MoveL Offs(pOrigin,191.56,41.34,0.00),v40,z0,tPen\WObj:=wPaper;
    MoveL Offs(pOrigin,191.21,43.25,0.00),v40,z0,tPen\WObj:=wPaper;
    MoveL Offs(pOrigin,190.07,44.74,0.00),v40,z0,tPen\WObj:=wPaper;
    MoveL Offs(pOrigin,190.07,44.74,0.00),v40,z0,tPen\WObj:=wPaper;
    MoveL Offs(pOrigin,188.59,44.95,0.00),v40,z0,tPen\WObj:=wPaper;
    MoveL Offs(pOrigin,188.16,45.38,0.00),v40,z0,tPen\WObj:=wPaper;
    MoveL Offs(pOrigin,188.16,45.38,0.00),v40,z0,tPen\WObj:=wPaper;
    MoveL Offs(pOrigin,189.23,48.35,0.00),v40,z0,tPen\WObj:=wPaper;
    MoveL Offs(pOrigin,189.23,48.35,0.00),v40,z0,tPen\WObj:=wPaper;
    MoveL Offs(pOrigin,191.14,47.71,0.00),v40,z0,tPen\WObj:=wPaper;
    MoveL Offs(pOrigin,191.14,47.71,0.00),v40,z0,tPen\WObj:=wPaper;
    MoveL Offs(pOrigin,190.07,44.74,0.00),v40,fine,tPen\WObj:=wPaper;
    MoveL Offs(pOrigin,190.07,44.74,6.00),v60,z5,tPen\WObj:=wPaper;
    MoveL Offs(pOrigin,190.07,43.25,6.00),vTravel,z5,tPen\WObj:=wPaper;
    MoveL Offs(pOrigin,190.07,43.25,0.00),v60,z0,tPen\WObj:=wPaper;
    MoveL Offs(pOrigin,189.23,43.96,0.00),v40,z0,tPen\WObj:=wPaper;
    MoveL Offs(pOrigin,187.52,44.10,0.00),v40,z0,tPen\WObj:=wPaper;
    MoveL Offs(pOrigin,186.25,43.25,0.00),v40,fine,tPen\WObj:=wPaper;
    MoveL Offs(pOrigin,186.25,43.25,6.00),v60,z5,tPen\WObj:=wPaper;
    MoveL Offs(pOrigin,188.16,45.38,6.00),vTravel,z5,tPen\WObj:=wPaper;
    MoveL Offs(pOrigin,188.16,45.38,0.00),v60,z0,tPen\WObj:=wPaper;
    MoveL Offs(pOrigin,186.25,44.53,0.00),v40,z0,tPen\WObj:=wPaper;
    MoveL Offs(pOrigin,185.12,43.04,0.00),v40,z0,tPen\WObj:=wPaper;
    MoveL Offs(pOrigin,184.76,41.34,0.00),v40,z0,tPen\WObj:=wPaper;
    MoveL Offs(pOrigin,185.19,39.21,0.00),v40,z0,tPen\WObj:=wPaper;
    MoveL Offs(pOrigin,185.19,39.21,0.00),v40,z0,tPen\WObj:=wPaper;
    MoveL Offs(pOrigin,187.10,38.15,0.00),v40,z0,tPen\WObj:=wPaper;
    MoveL Offs(pOrigin,189.23,37.94,0.00),v40,fine,tPen\WObj:=wPaper;
    MoveL Offs(pOrigin,189.23,37.94,6.00),v60,z5,tPen\WObj:=wPaper;
    MoveL Offs(pOrigin,185.19,39.21,6.00),vTravel,z5,tPen\WObj:=wPaper;
    MoveL Offs(pOrigin,185.19,39.21,0.00),v60,z0,tPen\WObj:=wPaper;
    MoveL Offs(pOrigin,181.57,40.20,0.00),v40,z0,tPen\WObj:=wPaper;
    MoveL Offs(pOrigin,179.24,41.34,0.00),v40,fine,tPen\WObj:=wPaper;
    MoveL Offs(pOrigin,179.24,41.34,6.00),v60,z5,tPen\WObj:=wPaper;
    MoveL Offs(pOrigin,183.70,50.90,6.00),vTravel,z5,tPen\WObj:=wPaper;
    MoveL Offs(pOrigin,183.70,50.90,0.00),v60,z0,tPen\WObj:=wPaper;
    MoveL Offs(pOrigin,184.12,50.69,0.00),v40,z0,tPen\WObj:=wPaper;
    MoveL Offs(pOrigin,183.70,50.90,0.00),v40,fine,tPen\WObj:=wPaper;
    MoveL Offs(pOrigin,183.70,50.90,6.00),v60,z5,tPen\WObj:=wPaper;
    MoveL Offs(pOrigin,182.00,51.96,6.00),vTravel,z5,tPen\WObj:=wPaper;
    MoveL Offs(pOrigin,182.00,51.96,0.00),v60,z0,tPen\WObj:=wPaper;
    MoveL Offs(pOrigin,182.43,51.75,0.00),v40,z0,tPen\WObj:=wPaper;
    MoveL Offs(pOrigin,182.00,51.96,0.00),v40,z0,tPen\WObj:=wPaper;
    MoveL Offs(pOrigin,181.57,52.17,0.00),v40,z0,tPen\WObj:=wPaper;
    MoveL Offs(pOrigin,184.34,50.40,0.00),v40,z0,tPen\WObj:=wPaper;
    MoveL Offs(pOrigin,189.23,48.35,0.00),v40,fine,tPen\WObj:=wPaper;
    MoveL Offs(pOrigin,189.23,48.35,6.00),v60,z5,tPen\WObj:=wPaper;
    MoveL Offs(pOrigin,191.14,47.71,6.00),vTravel,z5,tPen\WObj:=wPaper;
    MoveL Offs(pOrigin,191.14,47.71,0.00),v60,z0,tPen\WObj:=wPaper;
    MoveL Offs(pOrigin,201.76,44.53,0.00),v40,z0,tPen\WObj:=wPaper;
    MoveL Offs(pOrigin,208.99,42.83,0.00),v40,z0,tPen\WObj:=wPaper;
    MoveL Offs(pOrigin,209.62,42.19,0.00),v40,fine,tPen\WObj:=wPaper;
    MoveL Offs(pOrigin,209.62,42.19,6.00),v60,z5,tPen\WObj:=wPaper;
    MoveL Offs(pOrigin,213.02,42.19,6.00),vTravel,z5,tPen\WObj:=wPaper;
    MoveL Offs(pOrigin,213.02,42.19,0.00),v60,z0,tPen\WObj:=wPaper;
    MoveL Offs(pOrigin,214.51,41.55,0.00),v40,z0,tPen\WObj:=wPaper;
    MoveL Offs(pOrigin,217.49,41.34,0.00),v40,z0,tPen\WObj:=wPaper;
    MoveL Offs(pOrigin,218.12,41.55,0.00),v40,fine,tPen\WObj:=wPaper;
    MoveL Offs(pOrigin,218.12,41.55,6.00),v60,z5,tPen\WObj:=wPaper;
    MoveL Offs(pOrigin,214.51,43.67,6.00),vTravel,z5,tPen\WObj:=wPaper;
    MoveL Offs(pOrigin,214.51,43.67,0.00),v60,z0,tPen\WObj:=wPaper;
    MoveL Offs(pOrigin,214.94,44.10,0.00),v40,z0,tPen\WObj:=wPaper;
    MoveL Offs(pOrigin,214.51,43.67,0.00),v40,fine,tPen\WObj:=wPaper;
    MoveL Offs(pOrigin,214.51,43.67,6.00),v60,z5,tPen\WObj:=wPaper;
    MoveL Offs(pOrigin,213.45,42.61,6.00),vTravel,z5,tPen\WObj:=wPaper;
  ENDPROC

  PROC DrawPart55()
    MoveL Offs(pOrigin,213.45,42.61,0.00),v60,z0,tPen\WObj:=wPaper;
    MoveL Offs(pOrigin,213.66,43.04,0.00),v40,z0,tPen\WObj:=wPaper;
    MoveL Offs(pOrigin,213.45,42.61,0.00),v40,z0,tPen\WObj:=wPaper;
    MoveL Offs(pOrigin,213.02,42.19,0.00),v40,z0,tPen\WObj:=wPaper;
    MoveL Offs(pOrigin,209.84,42.12,0.00),v40,z0,tPen\WObj:=wPaper;
    MoveL Offs(pOrigin,208.35,40.06,0.00),v40,z0,tPen\WObj:=wPaper;
    MoveL Offs(pOrigin,204.74,37.65,0.00),v40,z0,tPen\WObj:=wPaper;
    MoveL Offs(pOrigin,201.98,36.73,0.00),v40,z0,tPen\WObj:=wPaper;
    MoveL Offs(pOrigin,201.34,36.03,0.00),v40,z0,tPen\WObj:=wPaper;
    MoveL Offs(pOrigin,201.34,36.03,0.00),v40,z0,tPen\WObj:=wPaper;
    MoveL Offs(pOrigin,202.19,35.17,0.00),v40,z0,tPen\WObj:=wPaper;
    MoveL Offs(pOrigin,228.96,33.90,0.00),v40,fine,tPen\WObj:=wPaper;
    MoveL Offs(pOrigin,228.96,33.90,6.00),v60,z5,tPen\WObj:=wPaper;
    MoveL Offs(pOrigin,250.00,31.99,6.00),vTravel,z5,tPen\WObj:=wPaper;
    MoveL Offs(pOrigin,250.00,31.99,0.00),v60,z0,tPen\WObj:=wPaper;
    MoveL Offs(pOrigin,250.85,32.84,0.00),v40,fine,tPen\WObj:=wPaper;
    MoveL Offs(pOrigin,250.85,32.84,6.00),v60,z5,tPen\WObj:=wPaper;
    MoveL Offs(pOrigin,251.27,30.08,6.00),vTravel,z5,tPen\WObj:=wPaper;
    MoveL Offs(pOrigin,251.27,30.08,0.00),v60,z0,tPen\WObj:=wPaper;
    MoveL Offs(pOrigin,251.56,30.71,0.00),v40,z0,tPen\WObj:=wPaper;
    MoveL Offs(pOrigin,252.34,31.21,0.00),v40,z0,tPen\WObj:=wPaper;
    MoveL Offs(pOrigin,254.68,31.77,0.00),v40,fine,tPen\WObj:=wPaper;
    MoveL Offs(pOrigin,254.68,31.77,6.00),v60,z5,tPen\WObj:=wPaper;
    MoveL Offs(pOrigin,254.68,30.29,6.00),vTravel,z5,tPen\WObj:=wPaper;
    MoveL Offs(pOrigin,254.68,30.29,0.00),v60,z0,tPen\WObj:=wPaper;
    MoveL Offs(pOrigin,251.91,29.72,0.00),v40,z0,tPen\WObj:=wPaper;
    MoveL Offs(pOrigin,251.27,30.08,0.00),v40,fine,tPen\WObj:=wPaper;
    MoveL Offs(pOrigin,251.27,30.08,6.00),v60,z5,tPen\WObj:=wPaper;
    MoveL Offs(pOrigin,255.74,29.23,6.00),vTravel,z5,tPen\WObj:=wPaper;
    MoveL Offs(pOrigin,255.74,29.23,0.00),v60,z0,tPen\WObj:=wPaper;
    MoveL Offs(pOrigin,255.10,29.86,0.00),v40,z0,tPen\WObj:=wPaper;
    MoveL Offs(pOrigin,255.74,29.23,0.00),v40,fine,tPen\WObj:=wPaper;
    MoveL Offs(pOrigin,255.74,29.23,6.00),v60,z5,tPen\WObj:=wPaper;
    MoveL Offs(pOrigin,259.14,35.81,6.00),vTravel,z5,tPen\WObj:=wPaper;
    MoveL Offs(pOrigin,259.14,35.81,0.00),v60,z0,tPen\WObj:=wPaper;
    MoveL Offs(pOrigin,259.56,36.03,0.00),v40,z0,tPen\WObj:=wPaper;
    MoveL Offs(pOrigin,259.14,35.81,0.00),v40,fine,tPen\WObj:=wPaper;
    MoveL Offs(pOrigin,259.14,35.81,6.00),v60,z5,tPen\WObj:=wPaper;
    MoveL Offs(pOrigin,249.36,48.14,6.00),vTravel,z5,tPen\WObj:=wPaper;
    MoveL Offs(pOrigin,249.36,48.14,0.00),v60,z0,tPen\WObj:=wPaper;
    MoveL Offs(pOrigin,250.21,48.99,0.00),v40,z0,tPen\WObj:=wPaper;
    MoveL Offs(pOrigin,249.36,48.14,0.00),v40,fine,tPen\WObj:=wPaper;
    MoveL Offs(pOrigin,249.36,48.14,6.00),v60,z5,tPen\WObj:=wPaper;
    MoveL Offs(pOrigin,252.55,51.33,6.00),vTravel,z5,tPen\WObj:=wPaper;
    MoveL Offs(pOrigin,252.55,51.33,0.00),v60,z0,tPen\WObj:=wPaper;
    MoveL Offs(pOrigin,252.98,51.75,0.00),v40,z0,tPen\WObj:=wPaper;
    MoveL Offs(pOrigin,252.55,51.33,0.00),v40,z0,tPen\WObj:=wPaper;
    MoveL Offs(pOrigin,253.19,51.96,0.00),v40,z0,tPen\WObj:=wPaper;
    MoveL Offs(pOrigin,253.82,52.60,0.00),v40,z0,tPen\WObj:=wPaper;
    MoveL Offs(pOrigin,253.19,51.96,0.00),v40,fine,tPen\WObj:=wPaper;
    MoveL Offs(pOrigin,253.19,51.96,6.00),v60,z5,tPen\WObj:=wPaper;
    MoveL Offs(pOrigin,255.10,53.88,6.00),vTravel,z5,tPen\WObj:=wPaper;
    MoveL Offs(pOrigin,255.10,53.88,0.00),v60,z0,tPen\WObj:=wPaper;
    MoveL Offs(pOrigin,255.52,54.30,0.00),v40,z0,tPen\WObj:=wPaper;
    MoveL Offs(pOrigin,255.10,53.88,0.00),v40,fine,tPen\WObj:=wPaper;
    MoveL Offs(pOrigin,255.10,53.88,6.00),v60,z5,tPen\WObj:=wPaper;
    MoveL Offs(pOrigin,248.51,65.56,6.00),vTravel,z5,tPen\WObj:=wPaper;
    MoveL Offs(pOrigin,248.51,65.56,0.00),v60,z0,tPen\WObj:=wPaper;
    MoveL Offs(pOrigin,250.64,66.62,0.00),v40,z0,tPen\WObj:=wPaper;
    MoveL Offs(pOrigin,251.27,68.75,0.00),v40,z0,tPen\WObj:=wPaper;
    MoveL Offs(pOrigin,250.21,70.66,0.00),v40,z0,tPen\WObj:=wPaper;
    MoveL Offs(pOrigin,248.09,71.30,0.00),v40,z0,tPen\WObj:=wPaper;
    MoveL Offs(pOrigin,246.18,70.03,0.00),v40,z0,tPen\WObj:=wPaper;
    MoveL Offs(pOrigin,245.54,68.11,0.00),v40,z0,tPen\WObj:=wPaper;
    MoveL Offs(pOrigin,246.39,66.48,0.00),v40,z0,tPen\WObj:=wPaper;
    MoveL Offs(pOrigin,248.51,65.56,0.00),v40,fine,tPen\WObj:=wPaper;
    MoveL Offs(pOrigin,248.51,65.56,6.00),v60,z5,tPen\WObj:=wPaper;
    MoveL Offs(pOrigin,260.84,66.62,6.00),vTravel,z5,tPen\WObj:=wPaper;
    MoveL Offs(pOrigin,260.84,66.62,0.00),v60,z0,tPen\WObj:=wPaper;
    MoveL Offs(pOrigin,265.94,71.94,0.00),v40,z0,tPen\WObj:=wPaper;
    MoveL Offs(pOrigin,269.55,76.40,0.00),v40,z0,tPen\WObj:=wPaper;
    MoveL Offs(pOrigin,271.67,79.80,0.00),v40,z0,tPen\WObj:=wPaper;
    MoveL Offs(pOrigin,272.74,80.44,0.00),v40,fine,tPen\WObj:=wPaper;
    MoveL Offs(pOrigin,272.74,80.44,6.00),v60,z5,tPen\WObj:=wPaper;
    MoveL Offs(pOrigin,267.85,79.38,6.00),vTravel,z5,tPen\WObj:=wPaper;
    MoveL Offs(pOrigin,267.85,79.38,0.00),v60,z0,tPen\WObj:=wPaper;
    MoveL Offs(pOrigin,263.39,73.64,0.00),v40,fine,tPen\WObj:=wPaper;
    MoveL Offs(pOrigin,263.39,73.64,6.00),v60,z5,tPen\WObj:=wPaper;
    MoveL Offs(pOrigin,265.30,71.51,6.00),vTravel,z5,tPen\WObj:=wPaper;
    MoveL Offs(pOrigin,265.30,71.51,0.00),v60,z0,tPen\WObj:=wPaper;
    MoveL Offs(pOrigin,265.94,72.15,0.00),v40,z0,tPen\WObj:=wPaper;
    MoveL Offs(pOrigin,265.30,71.51,0.00),v40,fine,tPen\WObj:=wPaper;
    MoveL Offs(pOrigin,265.30,71.51,6.00),v60,z5,tPen\WObj:=wPaper;
    MoveL Offs(pOrigin,266.58,73.00,6.00),vTravel,z5,tPen\WObj:=wPaper;
    MoveL Offs(pOrigin,266.58,73.00,0.00),v60,z0,tPen\WObj:=wPaper;
    MoveL Offs(pOrigin,267.21,73.64,0.00),v40,z0,tPen\WObj:=wPaper;
    MoveL Offs(pOrigin,266.58,73.00,0.00),v40,fine,tPen\WObj:=wPaper;
    MoveL Offs(pOrigin,266.58,73.00,6.00),v60,z5,tPen\WObj:=wPaper;
    MoveL Offs(pOrigin,267.21,78.31,6.00),vTravel,z5,tPen\WObj:=wPaper;
    MoveL Offs(pOrigin,267.21,78.31,0.00),v60,z0,tPen\WObj:=wPaper;
    MoveL Offs(pOrigin,267.64,78.95,0.00),v40,z0,tPen\WObj:=wPaper;
    MoveL Offs(pOrigin,267.21,78.31,0.00),v40,fine,tPen\WObj:=wPaper;
    MoveL Offs(pOrigin,267.21,78.31,6.00),v60,z5,tPen\WObj:=wPaper;
    MoveL Offs(pOrigin,275.29,65.78,6.00),vTravel,z5,tPen\WObj:=wPaper;
    MoveL Offs(pOrigin,275.29,65.78,0.00),v60,z0,tPen\WObj:=wPaper;
    MoveL Offs(pOrigin,274.44,64.85,0.00),v40,z0,tPen\WObj:=wPaper;
    MoveL Offs(pOrigin,270.19,62.80,0.00),v40,z0,tPen\WObj:=wPaper;
    MoveL Offs(pOrigin,270.19,62.80,0.00),v40,z0,tPen\WObj:=wPaper;
    MoveL Offs(pOrigin,270.68,61.74,0.00),v40,z0,tPen\WObj:=wPaper;
    MoveL Offs(pOrigin,272.38,59.83,0.00),v40,z0,tPen\WObj:=wPaper;
    MoveL Offs(pOrigin,273.45,57.70,0.00),v40,z0,tPen\WObj:=wPaper;
    MoveL Offs(pOrigin,274.01,55.36,0.00),v40,z0,tPen\WObj:=wPaper;
    MoveL Offs(pOrigin,274.01,55.36,0.00),v40,z0,tPen\WObj:=wPaper;
    MoveL Offs(pOrigin,278.90,56.99,0.00),v40,z0,tPen\WObj:=wPaper;
    MoveL Offs(pOrigin,281.38,58.41,0.00),v40,z0,tPen\WObj:=wPaper;
    MoveL Offs(pOrigin,281.88,59.19,0.00),v40,fine,tPen\WObj:=wPaper;
    MoveL Offs(pOrigin,281.88,59.19,6.00),v60,z5,tPen\WObj:=wPaper;
    MoveL Offs(pOrigin,280.17,57.91,6.00),vTravel,z5,tPen\WObj:=wPaper;
    MoveL Offs(pOrigin,280.17,57.91,0.00),v60,z0,tPen\WObj:=wPaper;
    MoveL Offs(pOrigin,280.60,58.12,0.00),v40,z0,tPen\WObj:=wPaper;
    MoveL Offs(pOrigin,280.17,57.91,0.00),v40,fine,tPen\WObj:=wPaper;
    MoveL Offs(pOrigin,280.17,57.91,6.00),v60,z5,tPen\WObj:=wPaper;
    MoveL Offs(pOrigin,273.38,64.50,6.00),vTravel,z5,tPen\WObj:=wPaper;
    MoveL Offs(pOrigin,273.38,64.50,0.00),v60,z0,tPen\WObj:=wPaper;
    MoveL Offs(pOrigin,273.80,64.71,0.00),v40,z0,tPen\WObj:=wPaper;
    MoveL Offs(pOrigin,273.38,64.50,0.00),v40,fine,tPen\WObj:=wPaper;
    MoveL Offs(pOrigin,273.38,64.50,6.00),v60,z5,tPen\WObj:=wPaper;
    MoveL Offs(pOrigin,274.23,43.25,6.00),vTravel,z5,tPen\WObj:=wPaper;
    MoveL Offs(pOrigin,274.23,43.25,0.00),v60,z0,tPen\WObj:=wPaper;
    MoveL Offs(pOrigin,274.65,43.46,0.00),v40,z0,tPen\WObj:=wPaper;
  ENDPROC

  PROC DrawPart56()
    MoveL Offs(pOrigin,274.23,43.25,0.00),v40,z0,tPen\WObj:=wPaper;
    MoveL Offs(pOrigin,273.38,42.83,0.00),v40,z0,tPen\WObj:=wPaper;
    MoveL Offs(pOrigin,273.80,43.04,0.00),v40,z0,tPen\WObj:=wPaper;
    MoveL Offs(pOrigin,273.38,42.83,0.00),v40,fine,tPen\WObj:=wPaper;
    MoveL Offs(pOrigin,273.38,42.83,6.00),v60,z5,tPen\WObj:=wPaper;
    MoveL Offs(pOrigin,314.17,30.71,6.00),vTravel,z5,tPen\WObj:=wPaper;
    MoveL Offs(pOrigin,314.17,30.71,0.00),v60,z0,tPen\WObj:=wPaper;
    MoveL Offs(pOrigin,314.81,31.99,0.00),v40,fine,tPen\WObj:=wPaper;
    MoveL Offs(pOrigin,314.81,31.99,6.00),v60,z5,tPen\WObj:=wPaper;
    MoveL Offs(pOrigin,314.17,27.74,6.00),vTravel,z5,tPen\WObj:=wPaper;
    MoveL Offs(pOrigin,314.17,27.74,0.00),v60,z0,tPen\WObj:=wPaper;
    MoveL Offs(pOrigin,315.24,27.10,0.00),v40,z0,tPen\WObj:=wPaper;
    MoveL Offs(pOrigin,316.73,26.89,0.00),v40,fine,tPen\WObj:=wPaper;
    MoveL Offs(pOrigin,316.73,26.89,6.00),v60,z5,tPen\WObj:=wPaper;
    MoveL Offs(pOrigin,343.08,29.86,6.00),vTravel,z5,tPen\WObj:=wPaper;
    MoveL Offs(pOrigin,343.08,29.86,0.00),v60,z0,tPen\WObj:=wPaper;
    MoveL Offs(pOrigin,343.08,30.08,0.00),v40,z0,tPen\WObj:=wPaper;
    MoveL Offs(pOrigin,342.86,29.65,0.00),v40,z0,tPen\WObj:=wPaper;
    MoveL Offs(pOrigin,343.29,29.44,0.00),v40,fine,tPen\WObj:=wPaper;
    MoveL Offs(pOrigin,343.29,29.44,6.00),v60,z5,tPen\WObj:=wPaper;
    MoveL Offs(pOrigin,352.21,90.43,6.00),vTravel,z5,tPen\WObj:=wPaper;
    MoveL Offs(pOrigin,352.21,90.43,0.00),v60,z0,tPen\WObj:=wPaper;
    MoveL Offs(pOrigin,351.65,90.64,0.00),v40,z0,tPen\WObj:=wPaper;
    MoveL Offs(pOrigin,351.08,91.84,0.00),v40,z0,tPen\WObj:=wPaper;
    MoveL Offs(pOrigin,349.88,92.34,0.00),v40,fine,tPen\WObj:=wPaper;
    MoveL Offs(pOrigin,349.88,92.34,6.00),v60,z5,tPen\WObj:=wPaper;
    MoveL Offs(pOrigin,348.81,95.31,6.00),vTravel,z5,tPen\WObj:=wPaper;
    MoveL Offs(pOrigin,348.81,95.31,0.00),v60,z0,tPen\WObj:=wPaper;
    MoveL Offs(pOrigin,348.60,95.74,0.00),v40,z0,tPen\WObj:=wPaper;
    MoveL Offs(pOrigin,348.81,95.31,0.00),v40,fine,tPen\WObj:=wPaper;
    MoveL Offs(pOrigin,348.81,95.31,6.00),v60,z5,tPen\WObj:=wPaper;
    MoveL Offs(pOrigin,352.00,103.81,6.00),vTravel,z5,tPen\WObj:=wPaper;
    MoveL Offs(pOrigin,352.00,103.81,0.00),v60,z0,tPen\WObj:=wPaper;
    MoveL Offs(pOrigin,353.27,105.09,0.00),v40,z0,tPen\WObj:=wPaper;
    MoveL Offs(pOrigin,352.00,103.81,0.00),v40,fine,tPen\WObj:=wPaper;
    MoveL Offs(pOrigin,352.00,103.81,6.00),v60,z5,tPen\WObj:=wPaper;
    MoveL Offs(pOrigin,347.11,105.30,6.00),vTravel,z5,tPen\WObj:=wPaper;
    MoveL Offs(pOrigin,347.11,105.30,0.00),v60,z0,tPen\WObj:=wPaper;
    MoveL Offs(pOrigin,347.54,105.51,0.00),v40,z0,tPen\WObj:=wPaper;
    MoveL Offs(pOrigin,347.11,105.30,0.00),v40,fine,tPen\WObj:=wPaper;
    MoveL Offs(pOrigin,347.11,105.30,6.00),v60,z5,tPen\WObj:=wPaper;
    MoveL Offs(pOrigin,358.59,105.09,6.00),vTravel,z5,tPen\WObj:=wPaper;
    MoveL Offs(pOrigin,358.59,105.09,0.00),v60,z0,tPen\WObj:=wPaper;
    MoveL Offs(pOrigin,361.56,106.43,0.00),v40,z0,tPen\WObj:=wPaper;
    MoveL Offs(pOrigin,366.24,107.85,0.00),v40,z0,tPen\WObj:=wPaper;
    MoveL Offs(pOrigin,372.83,108.70,0.00),v40,z0,tPen\WObj:=wPaper;
    MoveL Offs(pOrigin,381.54,108.28,0.00),v40,z0,tPen\WObj:=wPaper;
    MoveL Offs(pOrigin,386.85,107.21,0.00),v40,z0,tPen\WObj:=wPaper;
    MoveL Offs(pOrigin,391.31,105.72,0.00),v40,z0,tPen\WObj:=wPaper;
    MoveL Offs(pOrigin,390.89,105.94,0.00),v40,z0,tPen\WObj:=wPaper;
    MoveL Offs(pOrigin,391.31,105.72,0.00),v40,z0,tPen\WObj:=wPaper;
    MoveL Offs(pOrigin,390.89,105.94,0.00),v40,fine,tPen\WObj:=wPaper;
    MoveL Offs(pOrigin,390.89,105.94,6.00),v60,z5,tPen\WObj:=wPaper;
    MoveL Offs(pOrigin,396.62,108.49,6.00),vTravel,z5,tPen\WObj:=wPaper;
    MoveL Offs(pOrigin,396.62,108.49,0.00),v60,z0,tPen\WObj:=wPaper;
    MoveL Offs(pOrigin,395.77,109.20,0.00),v40,z0,tPen\WObj:=wPaper;
    MoveL Offs(pOrigin,391.10,111.32,0.00),v40,z0,tPen\WObj:=wPaper;
    MoveL Offs(pOrigin,384.94,113.16,0.00),v40,z0,tPen\WObj:=wPaper;
    MoveL Offs(pOrigin,383.45,113.16,0.00),v40,fine,tPen\WObj:=wPaper;
    MoveL Offs(pOrigin,383.45,113.16,6.00),v60,z5,tPen\WObj:=wPaper;
    MoveL Offs(pOrigin,397.26,108.28,6.00),vTravel,z5,tPen\WObj:=wPaper;
    MoveL Offs(pOrigin,397.26,108.28,0.00),v60,z0,tPen\WObj:=wPaper;
    MoveL Offs(pOrigin,399.60,106.50,0.00),v40,z0,tPen\WObj:=wPaper;
    MoveL Offs(pOrigin,400.88,106.15,0.00),v40,fine,tPen\WObj:=wPaper;
    MoveL Offs(pOrigin,400.88,106.15,6.00),v60,z5,tPen\WObj:=wPaper;
    MoveL Offs(pOrigin,401.51,105.09,6.00),vTravel,z5,tPen\WObj:=wPaper;
    MoveL Offs(pOrigin,401.51,105.09,0.00),v60,z0,tPen\WObj:=wPaper;
    MoveL Offs(pOrigin,401.30,105.51,0.00),v40,z0,tPen\WObj:=wPaper;
    MoveL Offs(pOrigin,401.51,105.09,0.00),v40,fine,tPen\WObj:=wPaper;
    MoveL Offs(pOrigin,401.51,105.09,6.00),v60,z5,tPen\WObj:=wPaper;
    MoveL Offs(pOrigin,347.54,138.02,6.00),vTravel,z5,tPen\WObj:=wPaper;
    MoveL Offs(pOrigin,347.54,138.02,0.00),v60,z0,tPen\WObj:=wPaper;
    MoveL Offs(pOrigin,340.10,132.93,0.00),v40,z0,tPen\WObj:=wPaper;
    MoveL Offs(pOrigin,336.70,130.16,0.00),v40,z0,tPen\WObj:=wPaper;
    MoveL Offs(pOrigin,333.94,127.40,0.00),v40,z0,tPen\WObj:=wPaper;
    MoveL Offs(pOrigin,334.58,126.97,0.00),v40,z0,tPen\WObj:=wPaper;
    MoveL Offs(pOrigin,343.92,129.74,0.00),v40,z0,tPen\WObj:=wPaper;
    MoveL Offs(pOrigin,344.70,129.67,0.00),v40,z0,tPen\WObj:=wPaper;
    MoveL Offs(pOrigin,345.20,126.76,0.00),v40,z0,tPen\WObj:=wPaper;
    MoveL Offs(pOrigin,345.20,120.39,0.00),v40,z0,tPen\WObj:=wPaper;
    MoveL Offs(pOrigin,344.92,118.90,0.00),v40,z0,tPen\WObj:=wPaper;
    MoveL Offs(pOrigin,344.35,118.40,0.00),v40,z0,tPen\WObj:=wPaper;
    MoveL Offs(pOrigin,325.86,112.95,0.00),v40,z0,tPen\WObj:=wPaper;
    MoveL Offs(pOrigin,296.75,105.72,0.00),v40,z0,tPen\WObj:=wPaper;
    MoveL Offs(pOrigin,293.99,105.94,0.00),v40,z0,tPen\WObj:=wPaper;
    MoveL Offs(pOrigin,293.99,105.94,0.00),v40,z0,tPen\WObj:=wPaper;
    MoveL Offs(pOrigin,292.92,103.39,0.00),v40,z0,tPen\WObj:=wPaper;
    MoveL Offs(pOrigin,291.86,98.07,0.00),v40,fine,tPen\WObj:=wPaper;
    MoveL Offs(pOrigin,291.86,98.07,6.00),v60,z5,tPen\WObj:=wPaper;
    MoveL Offs(pOrigin,293.99,105.94,6.00),vTravel,z5,tPen\WObj:=wPaper;
    MoveL Offs(pOrigin,293.99,105.94,0.00),v60,z0,tPen\WObj:=wPaper;
    MoveL Offs(pOrigin,295.26,111.04,0.00),v40,z0,tPen\WObj:=wPaper;
    MoveL Offs(pOrigin,296.89,116.14,0.00),v40,z0,tPen\WObj:=wPaper;
    MoveL Offs(pOrigin,297.39,116.78,0.00),v40,fine,tPen\WObj:=wPaper;
    MoveL Offs(pOrigin,297.39,116.78,6.00),v60,z5,tPen\WObj:=wPaper;
    MoveL Offs(pOrigin,301.85,115.29,6.00),vTravel,z5,tPen\WObj:=wPaper;
    MoveL Offs(pOrigin,301.85,115.29,0.00),v60,z0,tPen\WObj:=wPaper;
    MoveL Offs(pOrigin,341.80,126.12,0.00),v40,fine,tPen\WObj:=wPaper;
    MoveL Offs(pOrigin,341.80,126.12,6.00),v60,z5,tPen\WObj:=wPaper;
    MoveL Offs(pOrigin,335.00,128.68,6.00),vTravel,z5,tPen\WObj:=wPaper;
    MoveL Offs(pOrigin,335.00,128.68,0.00),v60,z0,tPen\WObj:=wPaper;
    MoveL Offs(pOrigin,335.42,129.10,0.00),v40,z0,tPen\WObj:=wPaper;
    MoveL Offs(pOrigin,335.00,128.68,0.00),v40,fine,tPen\WObj:=wPaper;
    MoveL Offs(pOrigin,335.00,128.68,6.00),v60,z5,tPen\WObj:=wPaper;
    MoveL Offs(pOrigin,333.94,126.97,6.00),vTravel,z5,tPen\WObj:=wPaper;
    MoveL Offs(pOrigin,333.94,126.97,0.00),v60,z0,tPen\WObj:=wPaper;
    MoveL Offs(pOrigin,299.94,117.20,0.00),v40,z0,tPen\WObj:=wPaper;
    MoveL Offs(pOrigin,297.60,116.85,0.00),v40,z0,tPen\WObj:=wPaper;
    MoveL Offs(pOrigin,298.02,119.75,0.00),v40,z0,tPen\WObj:=wPaper;
    MoveL Offs(pOrigin,317.79,182.01,0.00),v40,z0,tPen\WObj:=wPaper;
    MoveL Offs(pOrigin,317.36,182.79,0.00),v40,z0,tPen\WObj:=wPaper;
    MoveL Offs(pOrigin,306.52,186.40,0.00),v40,z0,tPen\WObj:=wPaper;
    MoveL Offs(pOrigin,303.55,187.61,0.00),v40,z0,tPen\WObj:=wPaper;
    MoveL Offs(pOrigin,302.91,188.39,0.00),v40,fine,tPen\WObj:=wPaper;
    MoveL Offs(pOrigin,302.91,188.39,6.00),v60,z5,tPen\WObj:=wPaper;
    MoveL Offs(pOrigin,292.29,195.19,6.00),vTravel,z5,tPen\WObj:=wPaper;
    MoveL Offs(pOrigin,292.29,195.19,0.00),v60,z0,tPen\WObj:=wPaper;
    MoveL Offs(pOrigin,291.65,195.82,0.00),v40,z0,tPen\WObj:=wPaper;
    MoveL Offs(pOrigin,292.29,195.19,0.00),v40,fine,tPen\WObj:=wPaper;
    MoveL Offs(pOrigin,292.29,195.19,6.00),v60,z5,tPen\WObj:=wPaper;
  ENDPROC

  PROC DrawPart57()
    MoveL Offs(pOrigin,305.67,206.88,6.00),vTravel,z5,tPen\WObj:=wPaper;
    MoveL Offs(pOrigin,305.67,206.88,0.00),v60,z0,tPen\WObj:=wPaper;
    MoveL Offs(pOrigin,305.04,207.51,0.00),v40,z0,tPen\WObj:=wPaper;
    MoveL Offs(pOrigin,305.67,206.88,0.00),v40,fine,tPen\WObj:=wPaper;
    MoveL Offs(pOrigin,305.67,206.88,6.00),v60,z5,tPen\WObj:=wPaper;
    MoveL Offs(pOrigin,303.76,209.21,6.00),vTravel,z5,tPen\WObj:=wPaper;
    MoveL Offs(pOrigin,303.76,209.21,0.00),v60,z0,tPen\WObj:=wPaper;
    MoveL Offs(pOrigin,303.12,209.85,0.00),v40,z0,tPen\WObj:=wPaper;
    MoveL Offs(pOrigin,303.76,209.21,0.00),v40,fine,tPen\WObj:=wPaper;
    MoveL Offs(pOrigin,303.76,209.21,6.00),v60,z5,tPen\WObj:=wPaper;
    MoveL Offs(pOrigin,318.42,191.57,6.00),vTravel,z5,tPen\WObj:=wPaper;
    MoveL Offs(pOrigin,318.42,191.57,0.00),v60,z0,tPen\WObj:=wPaper;
    MoveL Offs(pOrigin,318.21,192.00,0.00),v40,z0,tPen\WObj:=wPaper;
    MoveL Offs(pOrigin,318.42,191.57,0.00),v40,fine,tPen\WObj:=wPaper;
    MoveL Offs(pOrigin,318.42,191.57,6.00),v60,z5,tPen\WObj:=wPaper;
    MoveL Offs(pOrigin,334.36,197.10,6.00),vTravel,z5,tPen\WObj:=wPaper;
    MoveL Offs(pOrigin,334.36,197.10,0.00),v60,z0,tPen\WObj:=wPaper;
    MoveL Offs(pOrigin,316.30,203.26,0.00),v40,z0,tPen\WObj:=wPaper;
    MoveL Offs(pOrigin,310.77,204.54,0.00),v40,z0,tPen\WObj:=wPaper;
    MoveL Offs(pOrigin,308.01,204.40,0.00),v40,z0,tPen\WObj:=wPaper;
    MoveL Offs(pOrigin,302.49,210.91,0.00),v40,z0,tPen\WObj:=wPaper;
    MoveL Offs(pOrigin,302.13,212.19,0.00),v40,z0,tPen\WObj:=wPaper;
    MoveL Offs(pOrigin,303.34,212.40,0.00),v40,z0,tPen\WObj:=wPaper;
    MoveL Offs(pOrigin,311.20,210.27,0.00),v40,z0,tPen\WObj:=wPaper;
    MoveL Offs(pOrigin,318.42,207.80,0.00),v40,z0,tPen\WObj:=wPaper;
    MoveL Offs(pOrigin,338.40,199.58,0.00),v40,z0,tPen\WObj:=wPaper;
    MoveL Offs(pOrigin,347.54,196.68,0.00),v40,z0,tPen\WObj:=wPaper;
    MoveL Offs(pOrigin,366.66,191.57,0.00),v40,z0,tPen\WObj:=wPaper;
    MoveL Offs(pOrigin,369.64,190.58,0.00),v40,z0,tPen\WObj:=wPaper;
    MoveL Offs(pOrigin,370.70,189.88,0.00),v40,fine,tPen\WObj:=wPaper;
    MoveL Offs(pOrigin,370.70,189.88,6.00),v60,z5,tPen\WObj:=wPaper;
    MoveL Offs(pOrigin,368.58,186.26,6.00),vTravel,z5,tPen\WObj:=wPaper;
    MoveL Offs(pOrigin,368.58,186.26,0.00),v60,z0,tPen\WObj:=wPaper;
    MoveL Offs(pOrigin,368.79,186.69,0.00),v40,z0,tPen\WObj:=wPaper;
    MoveL Offs(pOrigin,368.58,186.26,0.00),v40,fine,tPen\WObj:=wPaper;
    MoveL Offs(pOrigin,368.58,186.26,6.00),v60,z5,tPen\WObj:=wPaper;
    MoveL Offs(pOrigin,374.95,183.71,6.00),vTravel,z5,tPen\WObj:=wPaper;
    MoveL Offs(pOrigin,374.95,183.71,0.00),v60,z0,tPen\WObj:=wPaper;
    MoveL Offs(pOrigin,375.16,184.14,0.00),v40,z0,tPen\WObj:=wPaper;
    MoveL Offs(pOrigin,374.95,183.71,0.00),v40,fine,tPen\WObj:=wPaper;
    MoveL Offs(pOrigin,374.95,183.71,6.00),v60,z5,tPen\WObj:=wPaper;
    MoveL Offs(pOrigin,377.50,184.77,6.00),vTravel,z5,tPen\WObj:=wPaper;
    MoveL Offs(pOrigin,377.50,184.77,0.00),v60,z0,tPen\WObj:=wPaper;
    MoveL Offs(pOrigin,377.08,184.99,0.00),v40,z0,tPen\WObj:=wPaper;
    MoveL Offs(pOrigin,376.86,186.05,0.00),v40,z0,tPen\WObj:=wPaper;
    MoveL Offs(pOrigin,376.44,186.05,0.00),v40,fine,tPen\WObj:=wPaper;
    MoveL Offs(pOrigin,376.44,186.05,6.00),v60,z5,tPen\WObj:=wPaper;
    MoveL Offs(pOrigin,346.69,137.60,6.00),vTravel,z5,tPen\WObj:=wPaper;
    MoveL Offs(pOrigin,346.69,137.60,0.00),v60,z0,tPen\WObj:=wPaper;
    MoveL Offs(pOrigin,347.11,137.81,0.00),v40,z0,tPen\WObj:=wPaper;
    MoveL Offs(pOrigin,346.69,137.60,0.00),v40,fine,tPen\WObj:=wPaper;
    MoveL Offs(pOrigin,346.69,137.60,6.00),v60,z5,tPen\WObj:=wPaper;
    MoveL Offs(pOrigin,213.45,51.96,6.00),vTravel,z5,tPen\WObj:=wPaper;
    MoveL Offs(pOrigin,213.45,51.96,0.00),v60,z0,tPen\WObj:=wPaper;
    MoveL Offs(pOrigin,211.11,52.74,0.00),v40,z0,tPen\WObj:=wPaper;
    MoveL Offs(pOrigin,201.76,57.98,0.00),v40,z0,tPen\WObj:=wPaper;
    MoveL Offs(pOrigin,186.89,62.73,0.00),v40,z0,tPen\WObj:=wPaper;
    MoveL Offs(pOrigin,184.62,63.72,0.00),v40,z0,tPen\WObj:=wPaper;
    MoveL Offs(pOrigin,183.70,64.50,0.00),v40,fine,tPen\WObj:=wPaper;
    MoveL Offs(pOrigin,183.70,64.50,6.00),v60,z5,tPen\WObj:=wPaper;
    MoveL Offs(pOrigin,204.52,37.72,6.00),vTravel,z5,tPen\WObj:=wPaper;
    MoveL Offs(pOrigin,204.52,37.72,0.00),v60,z0,tPen\WObj:=wPaper;
    MoveL Offs(pOrigin,204.95,37.94,0.00),v40,z0,tPen\WObj:=wPaper;
    MoveL Offs(pOrigin,204.52,37.72,0.00),v40,fine,tPen\WObj:=wPaper;
    MoveL Offs(pOrigin,204.52,37.72,6.00),v60,z5,tPen\WObj:=wPaper;
    MoveL Offs(pOrigin,172.23,129.52,6.00),vTravel,z5,tPen\WObj:=wPaper;
    MoveL Offs(pOrigin,172.23,129.52,0.00),v60,z0,tPen\WObj:=wPaper;
    MoveL Offs(pOrigin,175.27,136.11,0.00),v40,z0,tPen\WObj:=wPaper;
    MoveL Offs(pOrigin,177.11,141.43,0.00),v40,z0,tPen\WObj:=wPaper;
    MoveL Offs(pOrigin,178.39,146.74,0.00),v40,z0,tPen\WObj:=wPaper;
    MoveL Offs(pOrigin,179.24,153.32,0.00),v40,z0,tPen\WObj:=wPaper;
    MoveL Offs(pOrigin,179.02,160.12,0.00),v40,z0,tPen\WObj:=wPaper;
    MoveL Offs(pOrigin,178.39,164.16,0.00),v40,z0,tPen\WObj:=wPaper;
    MoveL Offs(pOrigin,176.33,169.69,0.00),v40,z0,tPen\WObj:=wPaper;
    MoveL Offs(pOrigin,174.14,173.09,0.00),v40,z0,tPen\WObj:=wPaper;
    MoveL Offs(pOrigin,174.35,172.66,0.00),v40,z0,tPen\WObj:=wPaper;
    MoveL Offs(pOrigin,174.14,173.09,0.00),v40,z0,tPen\WObj:=wPaper;
    MoveL Offs(pOrigin,174.35,172.66,0.00),v40,fine,tPen\WObj:=wPaper;
    MoveL Offs(pOrigin,174.35,172.66,6.00),v60,z5,tPen\WObj:=wPaper;
    MoveL Offs(pOrigin,176.26,169.48,6.00),vTravel,z5,tPen\WObj:=wPaper;
    MoveL Offs(pOrigin,176.26,169.48,0.00),v60,z0,tPen\WObj:=wPaper;
    MoveL Offs(pOrigin,176.05,169.90,0.00),v40,z0,tPen\WObj:=wPaper;
    MoveL Offs(pOrigin,176.26,169.48,0.00),v40,fine,tPen\WObj:=wPaper;
    MoveL Offs(pOrigin,176.26,169.48,6.00),v60,z5,tPen\WObj:=wPaper;
    MoveL Offs(pOrigin,173.29,132.07,6.00),vTravel,z5,tPen\WObj:=wPaper;
    MoveL Offs(pOrigin,173.29,132.07,0.00),v60,z0,tPen\WObj:=wPaper;
    MoveL Offs(pOrigin,173.50,132.50,0.00),v40,z0,tPen\WObj:=wPaper;
    MoveL Offs(pOrigin,173.29,132.07,0.00),v40,fine,tPen\WObj:=wPaper;
    MoveL Offs(pOrigin,173.29,132.07,6.00),v60,z5,tPen\WObj:=wPaper;
  ENDPROC

ENDMODULE
